ACTION OpenStopper2_action:
ST03_515_Y72_5.MoveWork:=TRUE;		(* Übergabeposition Stopper 2 *)
END_ACTION

ACTION WaitForPartOnPos3_entry:
ProcessMessage02:='';
Delay(IN:=FALSE);
END_ACTION

ACTION WaitForPartOnPos3_action:
ProcessMessage02:='2IM4';						(*warte auf Teil Übergabeposition 3*)
END_ACTION

ACTION WaitForPartOnPos3_exit:
ProcessMessage02:='';
END_ACTION

ACTION CloseStopper2_action:
ST03_515_Y72_5.MoveInit:=TRUE;		(* Übergabeposition Stopper 2 *)
END_ACTION

ACTION OpenStopper3_action:
ST03_515_Y72_6.MoveWork:=TRUE;		(* Übergabeposition Stopper 3 *)
END_ACTION

ACTION WaitForPartOnPos4_entry:
ProcessMessage02:='';
Delay(IN:=FALSE);
END_ACTION

ACTION WaitForPartOnPos4_action:
ProcessMessage02:='2IM3';						(*warte auf Teil Übergabeposition 4*)
Delay(
	IN:=NOT ST03_513_B70_7.BitInToCheck AND	(* ISK auf Übergabeposition  1*)
		NOT ST03_514_B71_2.BitInToCheck AND	(* ISK auf Übergabeposition  2*)
		NOT ST03_514_B71_5.BitInToCheck AND	(* ISK auf Übergabeposition  3*)
		NOT ST03_514_B71_6.BitInToCheck		(* ISK auf Übergabeposition  4*),
	PT:=t#1s);
END_ACTION

ACTION WaitForPartOnPos4_exit:
ProcessMessage02:='';
Delay(IN:=FALSE);
END_ACTION

ACTION CloseStopper3_action:
ST03_515_Y72_6.MoveInit:=TRUE;		(* Übergabeposition Stopper 3 *)
END_ACTION

ACTION SeqEnd_action:
SFCTime:=TIME_TO_DINT(TIME()-SFCTimeStart);
State:=STATE_WAIT;
END_ACTION

TRANSITION .ActualArea:
Robot01.ActualArea <> 4
END_TRANSITION

TRANSITION Check_Part:
NOT ST03_513_B70_7.BitInToCheck OR	(* ISK auf Übergabeposition  1*)
NOT ST03_514_B71_2.BitInToCheck OR	(* ISK auf Übergabeposition  2*)
NOT ST03_514_B71_5.BitInToCheck OR	(* ISK auf Übergabeposition  3*)
NOT ST03_514_B71_6.BitInToCheck		(* ISK auf Übergabeposition  4*)
END_TRANSITION

TRANSITION PosEmpty:
NOT ST03_513_B70_4.BitInToCheck			 	(*  ISK anwesend am Stopper*)
END_TRANSITION

TRANSITION State Ok:
ST03_515_Y72_2.State=STATE_OK (* Führungsschiene  Zuführung Vereinzler AST/GST *)
END_TRANSITION

TRANSITION Part Ready:
ST03_513_B70_4.BitInToCheck	(*  ISK anwesend am Stopper*)
END_TRANSITION

TRANSITION PosFull:
ST03_513_B70_4.BitInToCheck			 	(*  ISK anwesend am Stopper*)
END_TRANSITION

TRANSITION State Ok:
ST03_515_Y72_2.State=STATE_OK (* Führungsschiene  Zuführung Vereinzler AST/GST *)
END_TRANSITION

TRANSITION Pos1Empty:
NOT ST03_513_B70_7.BitInToCheck AND 	(*  ISK auf Übergabeposition 1*)
Robot01.ActualArea <> 4
END_TRANSITION

TRANSITION State Ok:
ST03_515_Y72_3.State=STATE_OK 	(* Führungsschiene  Zuführung Stopper AST/GST *)
END_TRANSITION

TRANSITION Pos1 Ready:
ST03_513_B70_7.BitInToCheck 		 (* ISK auf Übergabeposition 1 *)
END_TRANSITION

TRANSITION Pos1Full:
ST03_513_B70_7.BitInToCheck 	(*  ISK auf Übergabeposition 1*)
END_TRANSITION

TRANSITION State Ok:
ST03_515_Y72_3.State=STATE_OK AND 	(* Führungsschiene  Zuführung Stopper AST/GST *)
ST03_515_Y72_2.State=STATE_OK (* Führungsschiene  Zuführung Vereinzler AST/GST *)
END_TRANSITION

TRANSITION Pos2Empty:
NOT ST03_514_B71_2.BitInToCheck  	(*  ISK auf Übergabeposition 2*)
END_TRANSITION

TRANSITION State Ok:
ST03_515_Y72_4.State=STATE_OK 	(* Übergabeposition Stopper 1 AST/GST *)
END_TRANSITION

TRANSITION Pos3Full:
ST03_514_B71_5.BitInToCheck	 	(*  ISK auf Übergabeposition 3*)
END_TRANSITION

TRANSITION Pos3Empty:
NOT ST03_514_B71_5.BitInToCheck  	(*  ISK auf Übergabeposition 3*)
END_TRANSITION

TRANSITION Pos2 Ready:
ST03_514_B71_2.BitInToCheck 		 (* ISK auf Übergabeposition 2 *)
END_TRANSITION

TRANSITION Pos2Full:
ST03_514_B71_2.BitInToCheck	 	(*  ISK auf Übergabeposition 2*)
END_TRANSITION

TRANSITION State Ok:
ST03_515_Y72_4.State=STATE_OK 	(* Übergabeposition Stopper 1 AST/GST *)
END_TRANSITION

TRANSITION Pos3Empty:
NOT ST03_514_B71_5.BitInToCheck  	(*  ISK auf Übergabeposition 3*)
END_TRANSITION

TRANSITION State Ok:
ST03_515_Y72_5.State=STATE_OK 	(* Übergabeposition Stopper 2 AST/GST *)
END_TRANSITION

TRANSITION Po4Full:
ST03_514_B71_6.BitInToCheck 		(*  ISK auf Übergabeposition 4*)
END_TRANSITION

TRANSITION Pos4Empty:
NOT ST03_514_B71_6.BitInToCheck  	(*  ISK auf Übergabeposition 4*)
END_TRANSITION

TRANSITION Pos3 Ready:
ST03_514_B71_5.BitInToCheck 	 (* ISK auf Übergabeposition 3 *)
END_TRANSITION

TRANSITION Pos3Full:
ST03_514_B71_5.BitInToCheck	 	(*  ISK auf Übergabeposition 3*)
END_TRANSITION

TRANSITION State Ok:
ST03_515_Y72_5.State=STATE_OK 	(* Übergabeposition Stopper 2 AST/GST *)
END_TRANSITION

TRANSITION Pos4Empty:
NOT ST03_514_B71_6.BitInToCheck  	(*  ISK auf Übergabeposition 4*)
END_TRANSITION

TRANSITION State Ok:
ST03_515_Y72_6.State=STATE_OK 	(* Übergabeposition Stopper 3 AST/GST *)
END_TRANSITION

TRANSITION Pos4 Ready:
ST03_514_B71_6.BitInToCheck  OR		 (* ISK auf Übergabeposition 4 *)
Delay.Q
END_TRANSITION

TRANSITION Po4Full:
ST03_514_B71_6.BitInToCheck 		(*  ISK auf Übergabeposition 4*)
END_TRANSITION

TRANSITION State Ok:
ST03_515_Y72_6.State=STATE_OK 	(* Übergabeposition Stopper 3 AST/GST *)
END_TRANSITION
END_PROGRAM

(* POU Stations/ST_03_Ruestsaetze/ST_03_SFCs/Zufuehrungen/ST03_7pol_Wendeeinheit, SFC *)
 PROGRAM ST03_7pol_Wendeeinheit
VAR_OUTPUT
	SFCCurrentPOU			: STRING:='ST03_7pol_Wendeeinheit';
	SFCCurrentStep			: STRING:='';
	FB_CurrentStepHistorie	: FB_CurrentStepHistorie;
	SFCTime					: DINT;
	State   				: StateObject	:= STATE_WAIT;
	Result  				: StateResult;
END_VAR
VAR_INPUT
	Start				:BOOL;
END_VAR
VAR
	MsgOK				: BOOL;
	MsgCancel			: BOOL;
	SFCRun				: BOOL;
	SFCTimeStart		: TIME;
	Delay				: TON;
	(* Userdefinded area *)
	WenderDone			: BOOL;
	OverrideHelp			:DINT;
END_VAR
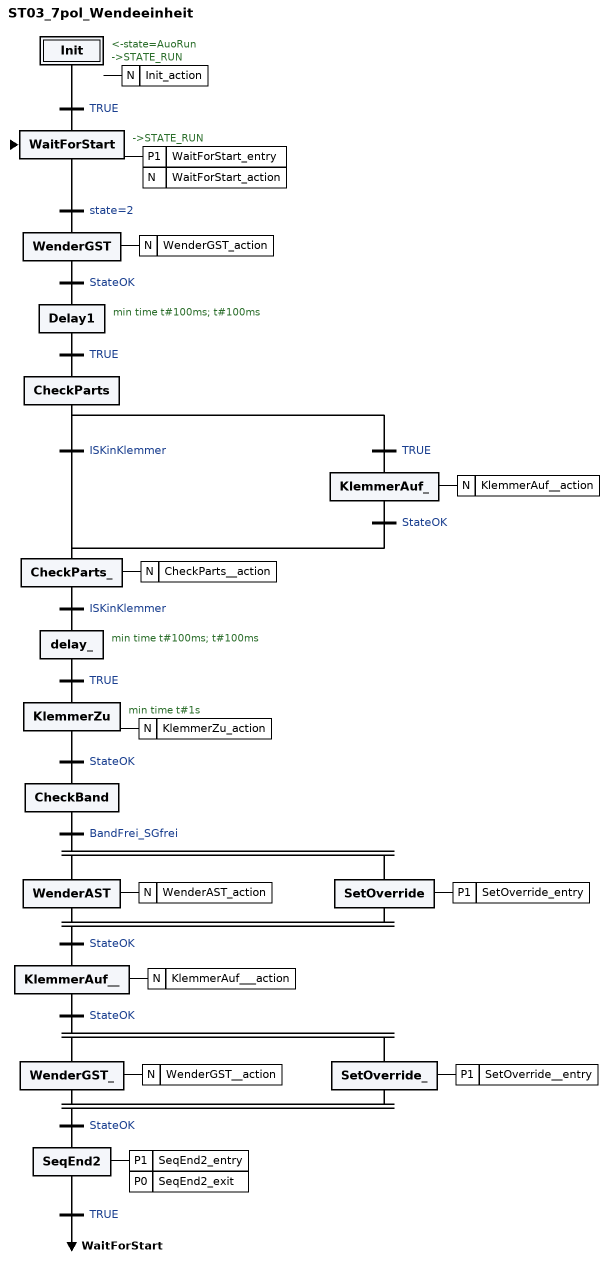
INITIAL_STEP Init: (* <-state=AuoRun / ->STATE_RUN *)
	Init_action(N);
END_STEP
TRANSITION FROM Init TO WaitForStart := TRUE;
END_TRANSITION
STEP WaitForStart: (* ->STATE_RUN *)
	WaitForStart_entry(P1);
	WaitForStart_action(N);
END_STEP
TRANSITION FROM WaitForStart TO WenderGST := state=2;
END_TRANSITION
STEP WenderGST:
	WenderGST_action(N);
END_STEP
TRANSITION FROM WenderGST TO Delay1 := StateOK;
END_TRANSITION
STEP Delay1: (* min time t#100ms; t#100ms *)
END_STEP
TRANSITION FROM Delay1 TO CheckParts := TRUE;
END_TRANSITION
STEP CheckParts:
END_STEP
TRANSITION FROM CheckParts TO CheckParts_ := ISKinKlemmer;
END_TRANSITION
TRANSITION FROM CheckParts TO KlemmerAuf_ := TRUE;
END_TRANSITION
STEP KlemmerAuf_:
	KlemmerAuf__action(N);
END_STEP
TRANSITION FROM KlemmerAuf_ TO CheckParts_ := StateOK;
END_TRANSITION
STEP CheckParts_:
	CheckParts__action(N);
END_STEP
TRANSITION FROM CheckParts_ TO delay_ := ISKinKlemmer;
END_TRANSITION
STEP delay_: (* min time t#100ms; t#100ms *)
END_STEP
TRANSITION FROM delay_ TO KlemmerZu := TRUE;
END_TRANSITION
STEP KlemmerZu: (* min time t#1s *)
	KlemmerZu_action(N);
END_STEP
TRANSITION FROM KlemmerZu TO CheckBand := StateOK;
END_TRANSITION
STEP CheckBand:
END_STEP
TRANSITION FROM CheckBand TO (WenderAST, SetOverride) := BandFrei_SGfrei;
END_TRANSITION
STEP WenderAST:
	WenderAST_action(N);
END_STEP
STEP SetOverride:
	SetOverride_entry(P1);
END_STEP
TRANSITION FROM (WenderAST, SetOverride) TO KlemmerAuf__ := StateOK;
END_TRANSITION
STEP KlemmerAuf__:
	KlemmerAuf___action(N);
END_STEP
TRANSITION FROM KlemmerAuf__ TO (WenderGST_, SetOverride_) := StateOK;
END_TRANSITION
STEP WenderGST_:
	WenderGST__action(N);
END_STEP
STEP SetOverride_:
	SetOverride__entry(P1);
END_STEP
TRANSITION FROM (WenderGST_, SetOverride_) TO SeqEnd2 := StateOK;
END_TRANSITION
STEP SeqEnd2:
	SeqEnd2_entry(P1);
	SeqEnd2_exit(P0);
END_STEP
TRANSITION FROM SeqEnd2 TO WaitForStart := TRUE;
END_TRANSITION

ACTION Init_action:
Start:=FALSE;
State:=STATE_WAIT;
MsgOK:=FALSE;
MsgCancel:=FALSE;
SFCRun:=FALSE;
Result:=RESULT_NON;
IF 	OverrideHelp <> 0 THEN
	MP.ST02.Override_Band:=OverrideHelp;
END_IF
END_ACTION

ACTION WaitForStart_entry:
;
END_ACTION

ACTION WaitForStart_action:
IF 	Start   THEN
	State:=STATE_RUN;
	Result:=RESULT_NON;
	SFCTimeStart:=TIME();
	Start:=FALSE;
	WenderDone:=FALSE;
ELSE
	State:=STATE_WAIT;
	MsgOK:=FALSE;
	MsgCancel:=FALSE;
	SFCRun:=FALSE;
END_IF
END_ACTION

ACTION WenderGST_action:
ST03_515_Y72_1.MoveInit:=TRUE;		(* Rinne schwenkern AST/GST *)
END_ACTION

ACTION KlemmerAuf__action:
ST03_515_Y72_0.MoveInit:=TRUE;		(* ISK Klemmer AST/GST *)
END_ACTION

ACTION CheckParts__action:
ProcessMessage01:='1IM6';						(*'warte auf Teil in Vereinzelung*)
END_ACTION

ACTION KlemmerZu_action:
ST03_515_Y72_0.MoveWork:=TRUE;		(* ISK Klemmer AST/GST *)
END_ACTION

ACTION WenderAST_action:
ST03_515_Y72_1.MoveWork:=TRUE;		(* Rinne schwenkern AST/GST *)
END_ACTION

ACTION SetOverride_entry:
IF 	MP.ST02.Override_Band > 10 THEN
	OverrideHelp:=MP.ST02.Override_Band;
	MP.ST02.Override_Band:= 0;
END_IF
END_ACTION

ACTION KlemmerAuf___action:
ST03_515_Y72_0.MoveInit:=TRUE;
END_ACTION

ACTION WenderGST__action:
ST03_515_Y72_1.MoveInit:=TRUE;		(* Rinne schwenkern AST/GST *)
END_ACTION

ACTION SetOverride__entry:
MP.ST02.Override_Band:=OverrideHelp;
END_ACTION

ACTION SeqEnd2_entry:
WenderDone:=TRUE;
END_ACTION

ACTION SeqEnd2_exit:
WenderDone:=FALSE;
END_ACTION

TRANSITION StateOK:
ST03_515_Y72_1.State = STATE_OK			 (* Rinne schwenkern AST/GST *)
AND gTipImp
END_TRANSITION

TRANSITION ISKinKlemmer:
ST03_512_XG1.BitInToCheck 	(* ISK in Klemmer *)
AND gTipImp
END_TRANSITION

TRANSITION StateOK:
ST03_515_Y72_0.State = STATE_OK		(*   ISK Klemmer AST/GST *)
AND gTipImp
END_TRANSITION

TRANSITION ISKinKlemmer:
ST03_512_XG1.BitInToCheck AND 	(* ISK in Klemmer *)
gTipImp
END_TRANSITION

TRANSITION StateOK:
ST03_515_Y72_0.State = STATE_OK			(* ISK Klemmer AST/GST *)
AND gTipImp
END_TRANSITION

TRANSITION BandFrei_SGfrei:
ST03_514_B71_7.BitInToCheck  	(* Führungsschiene frei zum schwenken *)
AND (ST00_73_K4.BitInToCheck OR ST02_S1_40K01.BitInToCheck)		(*Schnittstelle Freigabe von Spritzmaschine (nur für Anlagen ohne Rundtisch)*)
AND gTipImp
END_TRANSITION

TRANSITION StateOK:
ST03_515_Y72_1.State = STATE_OK 	(* Förderband  Zuführung Vereinzelner Wender AST/GST *)
AND gTipImp
END_TRANSITION

TRANSITION StateOK:
ST03_515_Y72_0.State = STATE_OK	(* ISK Klemmer AST/GST *)
AND gTipImp
END_TRANSITION

TRANSITION StateOK:
ST03_515_Y72_1.State = STATE_OK 	(* Rinne schwenkern AST/GST *)
AND gTipImp
END_TRANSITION
END_PROGRAM

(* POU Stations/ST_03_Ruestsaetze/ST_03_SFCs/Zufuehrungen/ST03_9pol_Wendeeinheit, SFC *)
 PROGRAM ST03_9pol_Wendeeinheit
VAR_OUTPUT
	SFCCurrentPOU			: STRING:='ST03_7pol_Wendeeinheit';
	SFCCurrentStep			: STRING:='';
	FB_CurrentStepHistorie	: FB_CurrentStepHistorie;
	SFCTime					: DINT;
	State   				: StateObject	:= STATE_WAIT;
	Result  				: StateResult;
END_VAR
VAR_INPUT
	Start				:BOOL;
END_VAR
VAR
	MsgOK				: BOOL;
	MsgCancel			: BOOL;
	SFCRun				: BOOL;
	SFCTimeStart		: TIME;
	Delay				: TON;
	(* Userdefinded area *)
	WenderDone			: BOOL;
	OverrideHelp			:DINT;
END_VAR
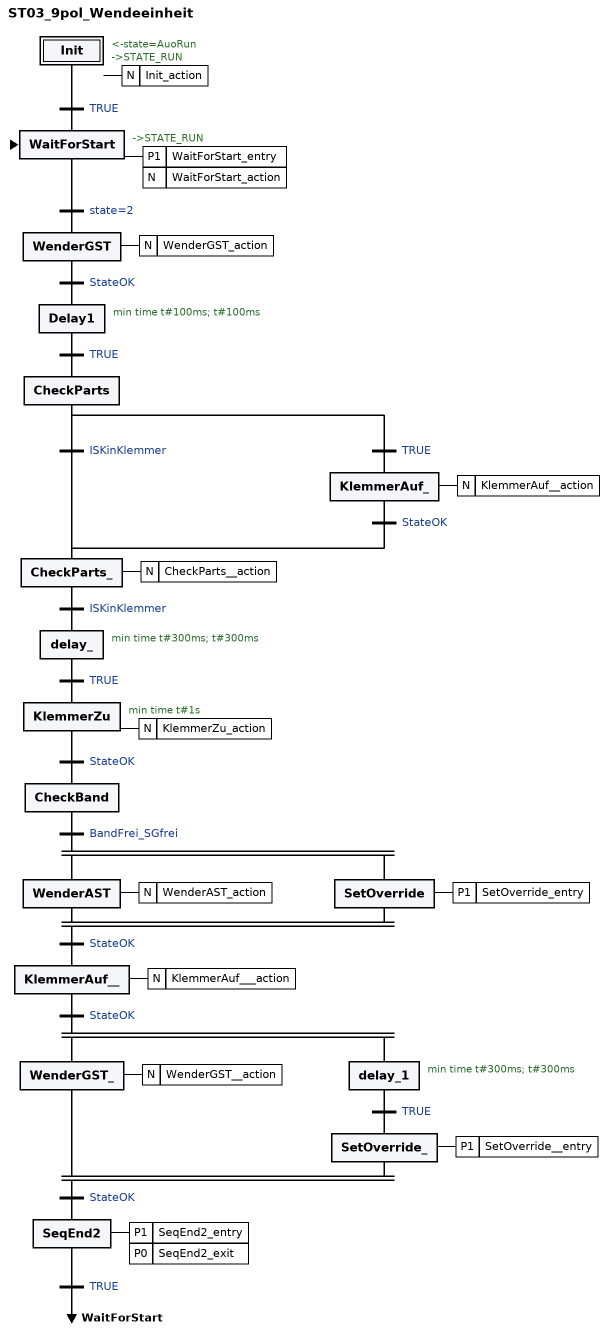
INITIAL_STEP Init: (* <-state=AuoRun / ->STATE_RUN *)
	Init_action(N);
END_STEP
TRANSITION FROM Init TO WaitForStart := TRUE;
END_TRANSITION
STEP WaitForStart: (* ->STATE_RUN *)
	WaitForStart_entry(P1);
	WaitForStart_action(N);
END_STEP
TRANSITION FROM WaitForStart TO WenderGST := state=2;
END_TRANSITION
STEP WenderGST:
	WenderGST_action(N);
END_STEP
TRANSITION FROM WenderGST TO Delay1 := StateOK;
END_TRANSITION
STEP Delay1: (* min time t#100ms; t#100ms *)
END_STEP
TRANSITION FROM Delay1 TO CheckParts := TRUE;
END_TRANSITION
STEP CheckParts:
END_STEP
TRANSITION FROM CheckParts TO CheckParts_ := ISKinKlemmer;
END_TRANSITION
TRANSITION FROM CheckParts TO KlemmerAuf_ := TRUE;
END_TRANSITION
STEP KlemmerAuf_:
	KlemmerAuf__action(N);
END_STEP
TRANSITION FROM KlemmerAuf_ TO CheckParts_ := StateOK;
END_TRANSITION
STEP CheckParts_:
	CheckParts__action(N);
END_STEP
TRANSITION FROM CheckParts_ TO delay_ := ISKinKlemmer;
END_TRANSITION
STEP delay_: (* min time t#300ms; t#300ms *)
END_STEP
TRANSITION FROM delay_ TO KlemmerZu := TRUE;
END_TRANSITION
STEP KlemmerZu: (* min time t#1s *)
	KlemmerZu_action(N);
END_STEP
TRANSITION FROM KlemmerZu TO CheckBand := StateOK;
END_TRANSITION
STEP CheckBand:
END_STEP
TRANSITION FROM CheckBand TO (WenderAST, SetOverride) := BandFrei_SGfrei;
END_TRANSITION
STEP WenderAST:
	WenderAST_action(N);
END_STEP
STEP SetOverride:
	SetOverride_entry(P1);
END_STEP
TRANSITION FROM (WenderAST, SetOverride) TO KlemmerAuf__ := StateOK;
END_TRANSITION
STEP KlemmerAuf__:
	KlemmerAuf___action(N);
END_STEP
TRANSITION FROM KlemmerAuf__ TO (WenderGST_, delay_1) := StateOK;
END_TRANSITION
STEP WenderGST_:
	WenderGST__action(N);
END_STEP
STEP delay_1: (* min time t#300ms; t#300ms *)
END_STEP
TRANSITION FROM delay_1 TO SetOverride_ := TRUE;
END_TRANSITION
STEP SetOverride_:
	SetOverride__entry(P1);
END_STEP
TRANSITION FROM (WenderGST_, SetOverride_) TO SeqEnd2 := StateOK;
END_TRANSITION
STEP SeqEnd2:
	SeqEnd2_entry(P1);
	SeqEnd2_exit(P0);
END_STEP
TRANSITION FROM SeqEnd2 TO WaitForStart := TRUE;
END_TRANSITION

ACTION Init_action:
Start:=FALSE;
State:=STATE_WAIT;
MsgOK:=FALSE;
MsgCancel:=FALSE;
SFCRun:=FALSE;
Result:=RESULT_NON;
IF 	OverrideHelp <> 0 THEN
	MP.ST02.Override_Band:=OverrideHelp;
END_IF
END_ACTION

ACTION WaitForStart_entry:
;
END_ACTION

ACTION WaitForStart_action:
IF 	Start   THEN
	State:=STATE_RUN;
	Result:=RESULT_NON;
	SFCTimeStart:=TIME();
	Start:=FALSE;
	WenderDone:=FALSE;
ELSE
	State:=STATE_WAIT;
	MsgOK:=FALSE;
	MsgCancel:=FALSE;
	SFCRun:=FALSE;
END_IF
END_ACTION

ACTION WenderGST_action:
ST03_515_Y72_1.MoveInit:=TRUE;		(* Rinne schwenkern AST/GST *)
END_ACTION

ACTION KlemmerAuf__action:
ST03_515_Y72_0.MoveInit:=TRUE;		(* ISK Klemmer AST/GST *)
END_ACTION

ACTION CheckParts__action:
ProcessMessage01:='1IM6';						(*'warte auf Teil in Vereinzelung*)
END_ACTION

ACTION KlemmerZu_action:
ST03_515_Y72_0.MoveWork:=TRUE;		(* ISK Klemmer AST/GST *)
END_ACTION

ACTION WenderAST_action:
ST03_515_Y72_1.MoveWork:=TRUE;		(* Rinne schwenkern AST/GST *)
END_ACTION

ACTION SetOverride_entry:
IF 	MP.ST02.Override_Band > 10 THEN
	OverrideHelp:=MP.ST02.Override_Band;
	MP.ST02.Override_Band:= 0;
END_IF
END_ACTION

ACTION KlemmerAuf___action:
ST03_515_Y72_0.MoveInit:=TRUE;
END_ACTION

ACTION WenderGST__action:
ST03_515_Y72_1.MoveInit:=TRUE;		(* Rinne schwenkern AST/GST *)
END_ACTION

ACTION SetOverride__entry:
MP.ST02.Override_Band:=OverrideHelp;
END_ACTION

ACTION SeqEnd2_entry:
WenderDone:=TRUE;
END_ACTION

ACTION SeqEnd2_exit:
WenderDone:=FALSE;
END_ACTION

TRANSITION StateOK:
ST03_515_Y72_1.State = STATE_OK			 (* Rinne schwenkern AST/GST *)
AND gTipImp
END_TRANSITION

TRANSITION ISKinKlemmer:
ST03_512_XG1.BitInToCheck 	(* ISK in Klemmer *)
AND gTipImp
END_TRANSITION

TRANSITION StateOK:
ST03_515_Y72_0.State = STATE_OK		(*   ISK Klemmer AST/GST *)
AND gTipImp
END_TRANSITION

TRANSITION ISKinKlemmer:
ST03_512_XG1.BitInToCheck AND 	(* ISK in Klemmer *)
gTipImp
END_TRANSITION

TRANSITION StateOK:
ST03_515_Y72_0.State = STATE_OK			(* ISK Klemmer AST/GST *)
AND gTipImp
END_TRANSITION

TRANSITION BandFrei_SGfrei:
ST03_514_B71_7.BitInToCheck  	(* Führungsschiene frei zum schwenken *)
AND (ST00_73_K4.BitInToCheck OR ST02_S1_40K01.BitInToCheck)		(*Schnittstelle Freigabe von Spritzmaschine (nur für Anlagen ohne Rundtisch)*)
AND gTipImp
END_TRANSITION

TRANSITION StateOK:
ST03_515_Y72_1.State = STATE_OK 	(* Förderband  Zuführung Vereinzelner Wender AST/GST *)
AND gTipImp
END_TRANSITION

TRANSITION StateOK:
ST03_515_Y72_0.State = STATE_OK	(* ISK Klemmer AST/GST *)
AND gTipImp
END_TRANSITION

TRANSITION StateOK:
ST03_515_Y72_1.State = STATE_OK 	(* Rinne schwenkern AST/GST *)
AND gTipImp
END_TRANSITION
END_PROGRAM

(* POU Stations/ST_03_Ruestsaetze/ST_03_SFCs/Zufuehrungen/ST03_88polAMG_Zufuehrung, SFC *)
 PROGRAM ST03_88polAMG_Zufuehrung
VAR_OUTPUT
	SFCCurrentPOU		: STRING:='ST03_88polAMG_Zufuehrung';
	SFCCurrentStep		: STRING:='';
	FB_CurrentStepHistorie: FB_CurrentStepHistorie;
	SFCTime				: DINT;
	State   			: StateObject	:= STATE_WAIT;
	Result  			: StateResult;
END_VAR
VAR_INPUT
	Start				:BOOL;
END_VAR
VAR
	MsgOK				: BOOL;
	MsgCancel			: BOOL;
	SFCRun				: BOOL;
	SFCTimeStart		: TIME;
	Delay				: TON;
	(* Userdefinded area *)

END_VAR
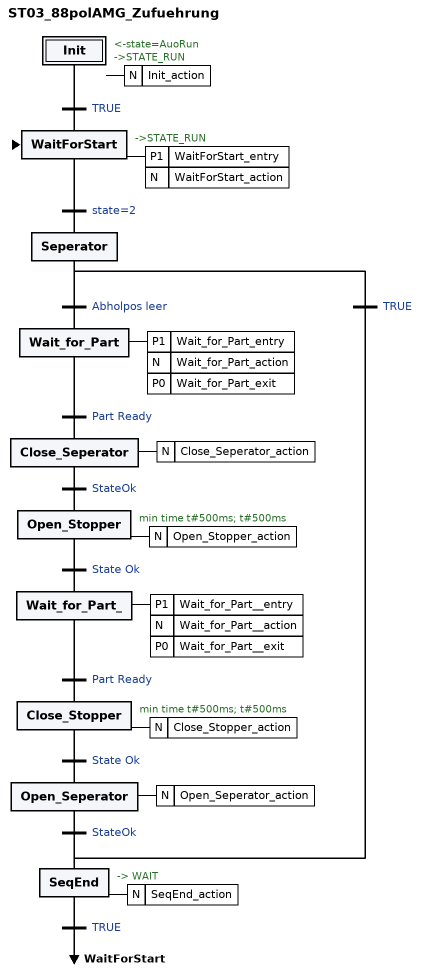
INITIAL_STEP Init: (* <-state=AuoRun / ->STATE_RUN *)
	Init_action(N);
END_STEP
TRANSITION FROM Init TO WaitForStart := TRUE;
END_TRANSITION
STEP WaitForStart: (* ->STATE_RUN *)
	WaitForStart_entry(P1);
	WaitForStart_action(N);
END_STEP
TRANSITION FROM WaitForStart TO Seperator := state=2;
END_TRANSITION
STEP Seperator:
END_STEP
TRANSITION FROM Seperator TO Wait_for_Part := Abholpos leer;
END_TRANSITION
TRANSITION FROM Seperator TO SeqEnd := TRUE;
END_TRANSITION
STEP Wait_for_Part:
	Wait_for_Part_entry(P1);
	Wait_for_Part_action(N);
	Wait_for_Part_exit(P0);
END_STEP
TRANSITION FROM Wait_for_Part TO Close_Seperator := Part Ready;
END_TRANSITION
STEP Close_Seperator:
	Close_Seperator_action(N);
END_STEP
TRANSITION FROM Close_Seperator TO Open_Stopper := StateOk;
END_TRANSITION
STEP Open_Stopper: (* min time t#500ms; t#500ms *)
	Open_Stopper_action(N);
END_STEP
TRANSITION FROM Open_Stopper TO Wait_for_Part_ := State Ok;
END_TRANSITION
STEP Wait_for_Part_:
	Wait_for_Part__entry(P1);
	Wait_for_Part__action(N);
	Wait_for_Part__exit(P0);
END_STEP
TRANSITION FROM Wait_for_Part_ TO Close_Stopper := Part Ready;
END_TRANSITION
STEP Close_Stopper: (* min time t#500ms; t#500ms *)
	Close_Stopper_action(N);
END_STEP
TRANSITION FROM Close_Stopper TO Open_Seperator := State Ok;
END_TRANSITION
STEP Open_Seperator:
	Open_Seperator_action(N);
END_STEP
TRANSITION FROM Open_Seperator TO SeqEnd := StateOk;
END_TRANSITION
STEP SeqEnd: (* -> WAIT *)
	SeqEnd_action(N);
END_STEP
TRANSITION FROM SeqEnd TO WaitForStart := TRUE;
END_TRANSITION

ACTION Init_action:
Start:=FALSE;
State:=STATE_WAIT;
MsgOK:=FALSE;
MsgCancel:=FALSE;
SFCRun:=FALSE;
Result:=RESULT_NON;
END_ACTION

ACTION WaitForStart_entry:
;
END_ACTION

ACTION WaitForStart_action:
IF 	Start   THEN
	State:=STATE_RUN;
	Result:=RESULT_NON;
	SFCTimeStart:=TIME();
	Start:=FALSE;
ELSE
	State:=STATE_WAIT;
	MsgOK:=FALSE;
	MsgCancel:=FALSE;
	SFCRun:=FALSE;
END_IF
END_ACTION

ACTION Wait_for_Part_entry:
ProcessMessage01:='';
Delay.IN:=FALSE;
Delay();
END_ACTION

ACTION Wait_for_Part_action:
ProcessMessage01:='1IM9';(*warte auf Teil in Stopper*)
Delay.IN:=ST03_521_B69_6.BitInToCheck; 		(*  ISK an stopper.*)
Delay.PT:=T#500ms;
Delay();
END_ACTION

ACTION Wait_for_Part_exit:
ProcessMessage01:='';
END_ACTION

ACTION Close_Seperator_action:
ST03_522_Y70_1.MoveWork:=TRUE;		(* Zuführung Vereinzler AST/GST *)
END_ACTION

ACTION Open_Stopper_action:
ST03_522_Y70_2.MoveWork:=TRUE;		(* Züführung Stopper AST/GST *)
END_ACTION

ACTION Wait_for_Part__entry:
ProcessMessage01:='';
Delay.IN:=FALSE;
Delay();
END_ACTION

ACTION Wait_for_Part__action:
ProcessMessage01:='1IM10';(*warte auf Teil in Abholposition*)
Delay.IN:=	ST03_Init_AbholPos.RoboPos31 OR
			ST03_Init_AbholPos.RoboPos35;
Delay.PT:=T#500ms;
Delay();
END_ACTION

ACTION Wait_for_Part__exit:
ProcessMessage01:='';
END_ACTION

ACTION Close_Stopper_action:
ST03_522_Y70_2.MoveInit:=TRUE;		(* Züführung Stopper AST/GST *)
END_ACTION

ACTION Open_Seperator_action:
ST03_522_Y70_1.MoveInit:=TRUE;		(* Zuführung Vereinzler AST/GST *)
END_ACTION

ACTION SeqEnd_action:
SFCTime:=TIME_TO_DINT(TIME()-SFCTimeStart);
State:=STATE_WAIT;
END_ACTION

TRANSITION Abholpos leer:
NOT  ST03_521_B69_7.BitInToCheck AND		(*  ISK Lageerkennung links*)
NOT  ST03_522_B70_0.BitInToCheck 		(*  ISK Lageerkennung rechts*)
END_TRANSITION

TRANSITION Part Ready:
Delay.Q AND
NOT ST03_521_B69_7.BitInToCheck	AND		(*  ISK Lageerkennung links*)
NOT ST03_522_B70_0.BitInToCheck	AND		(*  ISK Lageerkennung rechts*)
ST03_521_B69_6.BitInToCheck	AND				(*  ISK anwesend am Stoper*)
Robot01.ActualArea <> 4
END_TRANSITION

TRANSITION StateOk:
ST03_522_Y70_1.State=STATE_OK 	(* Zuführung Vereinzler AST/GST *)
END_TRANSITION

TRANSITION State Ok:
ST03_522_Y70_2.State=STATE_OK 	(* Züführung Stopper AST/GST *)
END_TRANSITION

TRANSITION Part Ready:
Delay.Q AND
Robot01.ActualArea <> 4
END_TRANSITION

TRANSITION State Ok:
ST03_522_Y70_2.State=STATE_OK 	(*Züführung Stopper AST/GST *)
END_TRANSITION

TRANSITION StateOk:
ST03_522_Y70_1.State=STATE_OK 	(* Zuführung Vereinzler AST/GST *)
END_TRANSITION
END_PROGRAM

(* POU Stations/ST_03_Ruestsaetze/ST_03_SFCs/Zufuehrungen/ST03_120pol_Zufuehrung, SFC *)
 PROGRAM ST03_120pol_Zufuehrung
VAR_OUTPUT
	SFCCurrentPOU		: STRING:='ST03_120pol_Zufuehrung';
	SFCCurrentStep		: STRING:='';
	FB_CurrentStepHistorie: FB_CurrentStepHistorie;
	SFCTime				: DINT;
	State   			: StateObject	:= STATE_WAIT;
	Result  			: StateResult;
END_VAR
VAR_INPUT
	Start				:BOOL;
END_VAR
VAR
	MsgOK				: BOOL;
	MsgCancel			: BOOL;
	SFCRun				: BOOL;
	SFCTimeStart		: TIME;
	Delay				: TON;
	(* Userdefinded area *)

END_VAR
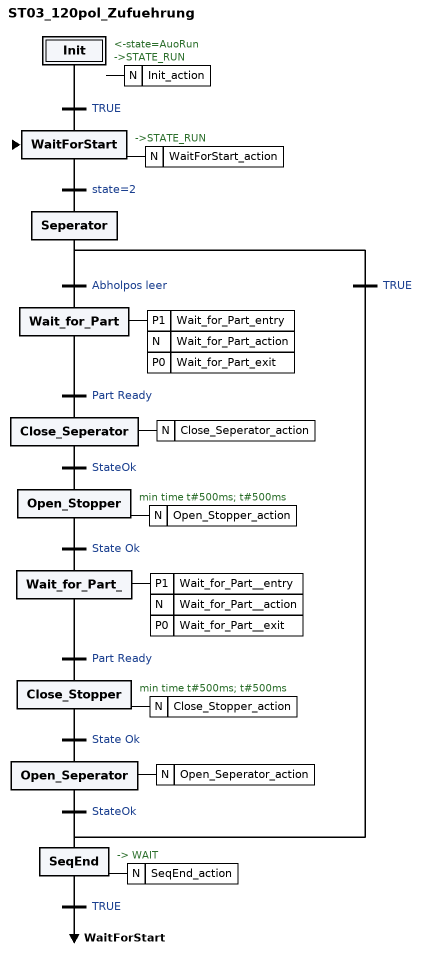
INITIAL_STEP Init: (* <-state=AuoRun / ->STATE_RUN *)
	Init_action(N);
END_STEP
TRANSITION FROM Init TO WaitForStart := TRUE;
END_TRANSITION
STEP WaitForStart: (* ->STATE_RUN *)
	WaitForStart_action(N);
END_STEP
TRANSITION FROM WaitForStart TO Seperator := state=2;
END_TRANSITION
STEP Seperator:
END_STEP
TRANSITION FROM Seperator TO Wait_for_Part := Abholpos leer;
END_TRANSITION
TRANSITION FROM Seperator TO SeqEnd := TRUE;
END_TRANSITION
STEP Wait_for_Part:
	Wait_for_Part_entry(P1);
	Wait_for_Part_action(N);
	Wait_for_Part_exit(P0);
END_STEP
TRANSITION FROM Wait_for_Part TO Close_Seperator := Part Ready;
END_TRANSITION
STEP Close_Seperator:
	Close_Seperator_action(N);
END_STEP
TRANSITION FROM Close_Seperator TO Open_Stopper := StateOk;
END_TRANSITION
STEP Open_Stopper: (* min time t#500ms; t#500ms *)
	Open_Stopper_action(N);
END_STEP
TRANSITION FROM Open_Stopper TO Wait_for_Part_ := State Ok;
END_TRANSITION
STEP Wait_for_Part_:
	Wait_for_Part__entry(P1);
	Wait_for_Part__action(N);
	Wait_for_Part__exit(P0);
END_STEP
TRANSITION FROM Wait_for_Part_ TO Close_Stopper := Part Ready;
END_TRANSITION
STEP Close_Stopper: (* min time t#500ms; t#500ms *)
	Close_Stopper_action(N);
END_STEP
TRANSITION FROM Close_Stopper TO Open_Seperator := State Ok;
END_TRANSITION
STEP Open_Seperator:
	Open_Seperator_action(N);
END_STEP
TRANSITION FROM Open_Seperator TO SeqEnd := StateOk;
END_TRANSITION
STEP SeqEnd: (* -> WAIT *)
	SeqEnd_action(N);
END_STEP
TRANSITION FROM SeqEnd TO WaitForStart := TRUE;
END_TRANSITION

ACTION Init_action:
Start:=FALSE;
State:=STATE_WAIT;
MsgOK:=FALSE;
MsgCancel:=FALSE;
SFCRun:=FALSE;
Result:=RESULT_NON;
END_ACTION

ACTION WaitForStart_action:
IF 	Start   THEN
	State:=STATE_RUN;
	Result:=RESULT_NON;
	SFCTimeStart:=TIME();
	Start:=FALSE;
ELSE
	State:=STATE_WAIT;
	MsgOK:=FALSE;
	MsgCancel:=FALSE;
	SFCRun:=FALSE;
END_IF
END_ACTION

ACTION Wait_for_Part_entry:
ProcessMessage01:='';
Delay.IN:=FALSE;
Delay();
END_ACTION

ACTION Wait_for_Part_action:
ProcessMessage01:='1IM9';(*warte auf Teil in Stopper*)
Delay.IN:=ST03_531_B69_6.BitInToCheck; 		(*  ISK an stopper.*)
Delay.PT:=T#500ms;
Delay();
END_ACTION

ACTION Wait_for_Part_exit:
ProcessMessage01:='';
END_ACTION

ACTION Close_Seperator_action:
ST03_532_Y70_1.MoveWork:=TRUE;		(*Zuführung Vereinzler AST/GST *)
END_ACTION

ACTION Open_Stopper_action:
ST03_532_Y70_2.MoveWork:=TRUE;		(* Züführung Stopper AST/GST *)
END_ACTION

ACTION Wait_for_Part__entry:
ProcessMessage01:='';
Delay.IN:=FALSE;
Delay();
END_ACTION

ACTION Wait_for_Part__action:
ProcessMessage01:='1IM10';(*warte auf Teil in Abholposition*)
Delay.IN:=	ST03_Init_AbholPos.RoboPos31 OR
			ST03_Init_AbholPos.RoboPos35;
Delay.PT:=T#500ms;
Delay();
END_ACTION

ACTION Wait_for_Part__exit:
ProcessMessage01:='';
END_ACTION

ACTION Close_Stopper_action:
ST03_532_Y70_2.MoveInit:=TRUE;		(* Züführung Stopper AST/GST *)
END_ACTION

ACTION Open_Seperator_action:
ST03_532_Y70_1.MoveInit:=TRUE;		(* Zuführung Vereinzler AST/GST *)
END_ACTION

ACTION SeqEnd_action:
SFCTime:=TIME_TO_DINT(TIME()-SFCTimeStart);
State:=STATE_WAIT;
END_ACTION

TRANSITION Abholpos leer:
NOT  ST03_531_B69_7.BitInToCheck AND	(*ISK rechts Lageerkennung*)
NOT ST03_532_B70_0.BitInToCheck		(*ISK links Lageerkennung*)
END_TRANSITION

TRANSITION Part Ready:
Delay.Q AND
NOT ST03_531_B69_7.BitInToCheck	AND		(*ISK rechts Lageerkennung*)
NOT ST03_532_B70_0.BitInToCheck	AND		(*ISK links Lageerkennung*)
ST03_531_B69_6.BitInToCheck	AND			(*ISK anwesend am Stoper*)
Robot01.ActualArea <> 4
END_TRANSITION

TRANSITION StateOk:
ST03_532_Y70_1.State=STATE_OK 	(* Zuführung Vereinzler AST/GST *)
END_TRANSITION

TRANSITION State Ok:
ST03_532_Y70_2.State=STATE_OK 	(* Züführung Stopper AST/GST *)
END_TRANSITION

TRANSITION Part Ready:
Delay.Q AND
Robot01.ActualArea <> 4
END_TRANSITION

TRANSITION State Ok:
ST03_532_Y70_2.State=STATE_OK 	(*Züführung Stopper AST/GST *)
END_TRANSITION

TRANSITION StateOk:
ST03_532_Y70_1.State=STATE_OK 	(* Zuführung Vereinzler AST/GST *)
END_TRANSITION
END_PROGRAM

(* POU Stations/ST_03_Ruestsaetze/ST_03_SFCs/Zufuehrungen/ST03_21pol_Zufuehrung, SFC *)
 PROGRAM ST03_21pol_Zufuehrung
VAR_OUTPUT
	SFCCurrentPOU		: STRING:='ST03_21pol_Zufuehrung';
	SFCCurrentStep		: STRING:='';
	FB_CurrentStepHistorie: FB_CurrentStepHistorie;
	SFCTime				: DINT;
	State   			: StateObject	:= STATE_WAIT;
	Result  			: StateResult;
END_VAR
VAR_INPUT
	Start				:BOOL;
END_VAR
VAR
	MsgOK				: BOOL;
	MsgCancel			: BOOL;
	SFCRun				: BOOL;
	SFCTimeStart		: TIME;
	Delay				: TON;
	(* Userdefinded area *)

END_VAR
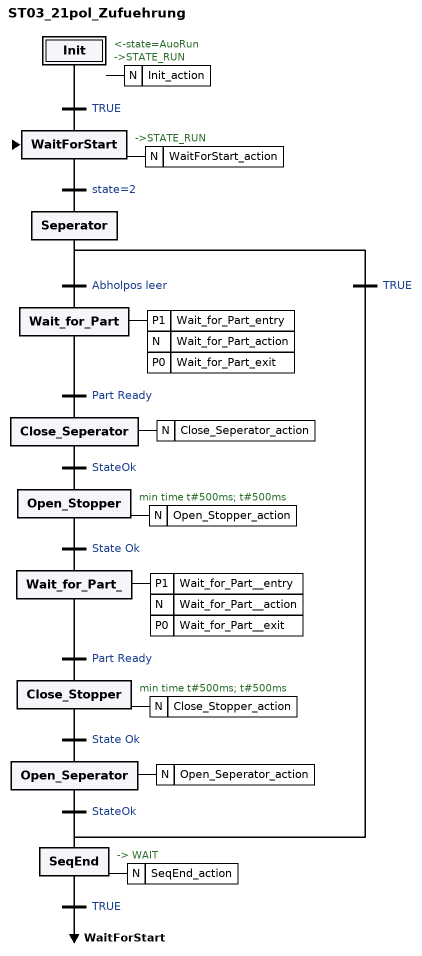
INITIAL_STEP Init: (* <-state=AuoRun / ->STATE_RUN *)
	Init_action(N);
END_STEP
TRANSITION FROM Init TO WaitForStart := TRUE;
END_TRANSITION
STEP WaitForStart: (* ->STATE_RUN *)
	WaitForStart_action(N);
END_STEP
TRANSITION FROM WaitForStart TO Seperator := state=2;
END_TRANSITION
STEP Seperator:
END_STEP
TRANSITION FROM Seperator TO Wait_for_Part := Abholpos leer;
END_TRANSITION
TRANSITION FROM Seperator TO SeqEnd := TRUE;
END_TRANSITION
STEP Wait_for_Part:
	Wait_for_Part_entry(P1);
	Wait_for_Part_action(N);
	Wait_for_Part_exit(P0);
END_STEP
TRANSITION FROM Wait_for_Part TO Close_Seperator := Part Ready;
END_TRANSITION
STEP Close_Seperator:
	Close_Seperator_action(N);
END_STEP
TRANSITION FROM Close_Seperator TO Open_Stopper := StateOk;
END_TRANSITION
STEP Open_Stopper: (* min time t#500ms; t#500ms *)
	Open_Stopper_action(N);
END_STEP
TRANSITION FROM Open_Stopper TO Wait_for_Part_ := State Ok;
END_TRANSITION
STEP Wait_for_Part_:
	Wait_for_Part__entry(P1);
	Wait_for_Part__action(N);
	Wait_for_Part__exit(P0);
END_STEP
TRANSITION FROM Wait_for_Part_ TO Close_Stopper := Part Ready;
END_TRANSITION
STEP Close_Stopper: (* min time t#500ms; t#500ms *)
	Close_Stopper_action(N);
END_STEP
TRANSITION FROM Close_Stopper TO Open_Seperator := State Ok;
END_TRANSITION
STEP Open_Seperator:
	Open_Seperator_action(N);
END_STEP
TRANSITION FROM Open_Seperator TO SeqEnd := StateOk;
END_TRANSITION
STEP SeqEnd: (* -> WAIT *)
	SeqEnd_action(N);
END_STEP
TRANSITION FROM SeqEnd TO WaitForStart := TRUE;
END_TRANSITION

ACTION Init_action:
Start:=FALSE;
State:=STATE_WAIT;
MsgOK:=FALSE;
MsgCancel:=FALSE;
SFCRun:=FALSE;
Result:=RESULT_NON;
END_ACTION

ACTION WaitForStart_action:
IF 	Start   THEN
	State:=STATE_RUN;
	Result:=RESULT_NON;
	SFCTimeStart:=TIME();
	Start:=FALSE;
ELSE
	State:=STATE_WAIT;
	MsgOK:=FALSE;
	MsgCancel:=FALSE;
	SFCRun:=FALSE;
END_IF
END_ACTION

ACTION Wait_for_Part_entry:
ProcessMessage01:='';
Delay.IN:=FALSE;
Delay();
END_ACTION

ACTION Wait_for_Part_action:
ProcessMessage01:='1IM9';(*warte auf Teil in Stopper*)
Delay.IN:=ST03_536_B69_6.BitInToCheck; 		(*  ISK an stopper.*)
Delay.PT:=T#500ms;
Delay();
END_ACTION

ACTION Wait_for_Part_exit:
ProcessMessage01:='';
END_ACTION

ACTION Close_Seperator_action:
ST03_537_Y70_1.MoveWork:=TRUE;		(*Zuführung Vereinzler AST/GST *)
END_ACTION

ACTION Open_Stopper_action:
ST03_537_Y70_2.MoveWork:=TRUE;		(* Züführung Stopper AST/GST *)
END_ACTION

ACTION Wait_for_Part__entry:
ProcessMessage01:='';
Delay.IN:=FALSE;
Delay();
END_ACTION

ACTION Wait_for_Part__action:
ProcessMessage01:='1IM10';(*warte auf Teil in Abholposition*)
Delay.IN:=	ST03_Init_AbholPos.RoboPos31 OR
			ST03_Init_AbholPos.RoboPos35;
Delay.PT:=T#500ms;
Delay();
END_ACTION

ACTION Wait_for_Part__exit:
ProcessMessage01:='';
END_ACTION

ACTION Close_Stopper_action:
ST03_537_Y70_2.MoveInit:=TRUE;		(* Züführung Stopper AST/GST *)
END_ACTION

ACTION Open_Seperator_action:
ST03_537_Y70_1.MoveInit:=TRUE;		(* Zuführung Vereinzler AST/GST *)
END_ACTION

ACTION SeqEnd_action:
SFCTime:=TIME_TO_DINT(TIME()-SFCTimeStart);
State:=STATE_WAIT;
END_ACTION

TRANSITION Abholpos leer:
NOT  ST03_536_B69_7.BitInToCheck		(*  ISK anwesend an Abholposition*)
END_TRANSITION

TRANSITION Part Ready:
Delay.Q AND
NOT ST03_536_B69_7.BitInToCheck	AND		(*ISK anwesend an Abholposition*)
NOT ST03_537_B70_0.BitInToCheck	AND		(*ISK Lageerkennung*)
ST03_536_B69_6.BitInToCheck	AND			(*ISK anwesend am Stoper*)
Robot01.ActualArea <> 4
END_TRANSITION

TRANSITION StateOk:
ST03_537_Y70_1.State=STATE_OK 	(* Zuführung Vereinzler AST/GST *)
END_TRANSITION

TRANSITION State Ok:
ST03_537_Y70_2.State=STATE_OK 	(* Züführung Stopper AST/GST *)
END_TRANSITION

TRANSITION Part Ready:
Delay.Q AND
Robot01.ActualArea <> 4
END_TRANSITION

TRANSITION State Ok:
ST03_537_Y70_2.State=STATE_OK 	(*Züführung Stopper AST/GST *)
END_TRANSITION

TRANSITION StateOk:
ST03_537_Y70_1.State=STATE_OK 	(* Zuführung Vereinzler AST/GST *)
END_TRANSITION
END_PROGRAM

(* POU Stations/ST_03_Ruestsaetze/ST_03_SFCs/Zufuehrungen/ST03_191pol_Zufuehrung, SFC *)
 PROGRAM ST03_191pol_Zufuehrung
VAR_OUTPUT
	SFCCurrentPOU		: STRING:='ST03_191pol_Zufuehrung';
	SFCCurrentStep		: STRING:='';
	FB_CurrentStepHistorie: FB_CurrentStepHistorie;
	SFCTime				: DINT;
	State   			: StateObject	:= STATE_WAIT;
	Result  			: StateResult;
END_VAR
VAR_INPUT
	Start				:BOOL;
END_VAR
VAR
	MsgOK				: BOOL;
	MsgCancel			: BOOL;
	SFCRun				: BOOL;
	SFCTimeStart		: TIME;
	Delay				: TON;
	(* Userdefinded area *)

END_VAR
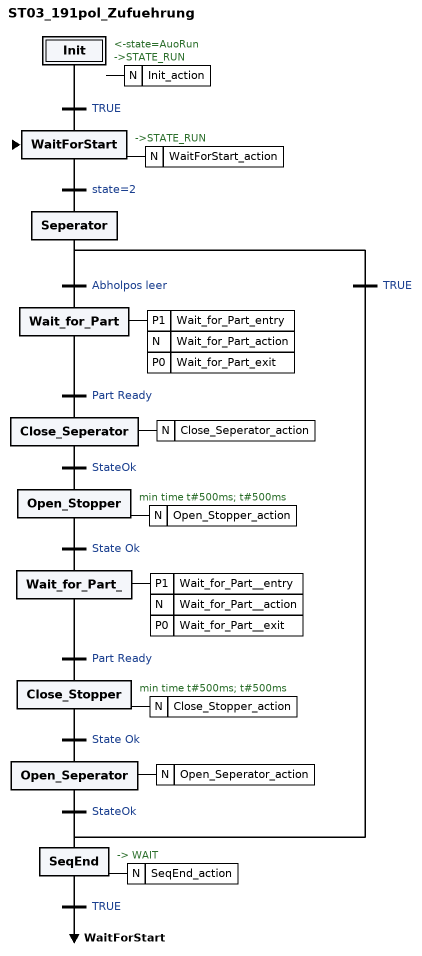
INITIAL_STEP Init: (* <-state=AuoRun / ->STATE_RUN *)
	Init_action(N);
END_STEP
TRANSITION FROM Init TO WaitForStart := TRUE;
END_TRANSITION
STEP WaitForStart: (* ->STATE_RUN *)
	WaitForStart_action(N);
END_STEP
TRANSITION FROM WaitForStart TO Seperator := state=2;
END_TRANSITION
STEP Seperator:
END_STEP
TRANSITION FROM Seperator TO Wait_for_Part := Abholpos leer;
END_TRANSITION
TRANSITION FROM Seperator TO SeqEnd := TRUE;
END_TRANSITION
STEP Wait_for_Part:
	Wait_for_Part_entry(P1);
	Wait_for_Part_action(N);
	Wait_for_Part_exit(P0);
END_STEP
TRANSITION FROM Wait_for_Part TO Close_Seperator := Part Ready;
END_TRANSITION
STEP Close_Seperator:
	Close_Seperator_action(N);
END_STEP
TRANSITION FROM Close_Seperator TO Open_Stopper := StateOk;
END_TRANSITION
STEP Open_Stopper: (* min time t#500ms; t#500ms *)
	Open_Stopper_action(N);
END_STEP
TRANSITION FROM Open_Stopper TO Wait_for_Part_ := State Ok;
END_TRANSITION
STEP Wait_for_Part_:
	Wait_for_Part__entry(P1);
	Wait_for_Part__action(N);
	Wait_for_Part__exit(P0);
END_STEP
TRANSITION FROM Wait_for_Part_ TO Close_Stopper := Part Ready;
END_TRANSITION
STEP Close_Stopper: (* min time t#500ms; t#500ms *)
	Close_Stopper_action(N);
END_STEP
TRANSITION FROM Close_Stopper TO Open_Seperator := State Ok;
END_TRANSITION
STEP Open_Seperator:
	Open_Seperator_action(N);
END_STEP
TRANSITION FROM Open_Seperator TO SeqEnd := StateOk;
END_TRANSITION
STEP SeqEnd: (* -> WAIT *)
	SeqEnd_action(N);
END_STEP
TRANSITION FROM SeqEnd TO WaitForStart := TRUE;
END_TRANSITION

ACTION Init_action:
Start:=FALSE;
State:=STATE_WAIT;
MsgOK:=FALSE;
MsgCancel:=FALSE;
SFCRun:=FALSE;
Result:=RESULT_NON;
END_ACTION

ACTION WaitForStart_action:
IF 	Start   THEN
	State:=STATE_RUN;
	Result:=RESULT_NON;
	SFCTimeStart:=TIME();
	Start:=FALSE;
ELSE
	State:=STATE_WAIT;
	MsgOK:=FALSE;
	MsgCancel:=FALSE;
	SFCRun:=FALSE;
END_IF
END_ACTION

ACTION Wait_for_Part_entry:
ProcessMessage01:='';
Delay.IN:=FALSE;
Delay();
END_ACTION

ACTION Wait_for_Part_action:
ProcessMessage01:='1IM9';(*warte auf Teil in Stopper*)
Delay.IN:=ST03_541_B69_6.BitInToCheck; 		(*  ISK an stopper.*)
Delay.PT:=T#500ms;
Delay();
END_ACTION

ACTION Wait_for_Part_exit:
ProcessMessage01:='';
END_ACTION

ACTION Close_Seperator_action:
ST03_542_Y70_1.MoveWork:=TRUE;		(*Zuführung Vereinzler AST/GST *)
END_ACTION

ACTION Open_Stopper_action:
ST03_542_Y70_2.MoveWork:=TRUE;		(* Züführung Stopper AST/GST *)
END_ACTION

ACTION Wait_for_Part__entry:
ProcessMessage01:='';
Delay.IN:=FALSE;
Delay();
END_ACTION

ACTION Wait_for_Part__action:
ProcessMessage01:='1IM10';(*warte auf Teil in Abholposition*)
Delay.IN:=	ST03_Init_AbholPos.RoboPos31 OR
			ST03_Init_AbholPos.RoboPos35;
Delay.PT:=T#500ms;
Delay();
END_ACTION

ACTION Wait_for_Part__exit:
ProcessMessage01:='';
END_ACTION

ACTION Close_Stopper_action:
ST03_542_Y70_2.MoveInit:=TRUE;		(* Züführung Stopper AST/GST *)
END_ACTION

ACTION Open_Seperator_action:
ST03_542_Y70_1.MoveInit:=TRUE;		(* Zuführung Vereinzler AST/GST *)
END_ACTION

ACTION SeqEnd_action:
SFCTime:=TIME_TO_DINT(TIME()-SFCTimeStart);
State:=STATE_WAIT;
END_ACTION

TRANSITION Abholpos leer:
NOT ST03_Init_AbholPos.RoboPos31 AND
NOT ST03_Init_AbholPos.RoboPos35
END_TRANSITION

TRANSITION Part Ready:
Delay.Q AND
NOT ST03_541_B69_7.BitInToCheck	AND		(*ISK links Lageerkennung*)
NOT ST03_542_B70_0.BitInToCheck	AND		(*ISK rechts Lageerkennung*)
ST03_541_B69_6.BitInToCheck	AND			(*ISK anwesend am Stoper*)
Robot01.ActualArea <> 4
END_TRANSITION

TRANSITION StateOk:
ST03_542_Y70_1.State=STATE_OK 	(* Zuführung Vereinzler AST/GST *)
END_TRANSITION

TRANSITION State Ok:
ST03_542_Y70_2.State=STATE_OK 	(* Züführung Stopper AST/GST *)
END_TRANSITION

TRANSITION Part Ready:
Delay.Q AND
Robot01.ActualArea <> 4
END_TRANSITION

TRANSITION State Ok:
ST03_542_Y70_2.State=STATE_OK 	(*Züführung Stopper AST/GST *)
END_TRANSITION

TRANSITION StateOk:
ST03_542_Y70_1.State=STATE_OK 	(* Zuführung Vereinzler AST/GST *)
END_TRANSITION
END_PROGRAM

(* POU Stations/ST_03_Ruestsaetze/ST_03_SFCs/Zufuehrungen/ST03_72pol_Zufuehrung, SFC *)
 PROGRAM ST03_72pol_Zufuehrung
VAR_OUTPUT
	SFCCurrentPOU		: STRING:='ST03_72pol_Zufuehrung';
	SFCCurrentStep		: STRING:='';
	FB_CurrentStepHistorie: FB_CurrentStepHistorie;
	SFCTime				: DINT;
	State   			: StateObject	:= STATE_WAIT;
	Result  			: StateResult;
END_VAR
VAR_INPUT
	Start				:BOOL;
END_VAR
VAR
	MsgOK				: BOOL;
	MsgCancel			: BOOL;
	SFCRun				: BOOL;
	SFCTimeStart		: TIME;
	Delay				: TON;
	(* Userdefinded area *)

END_VAR
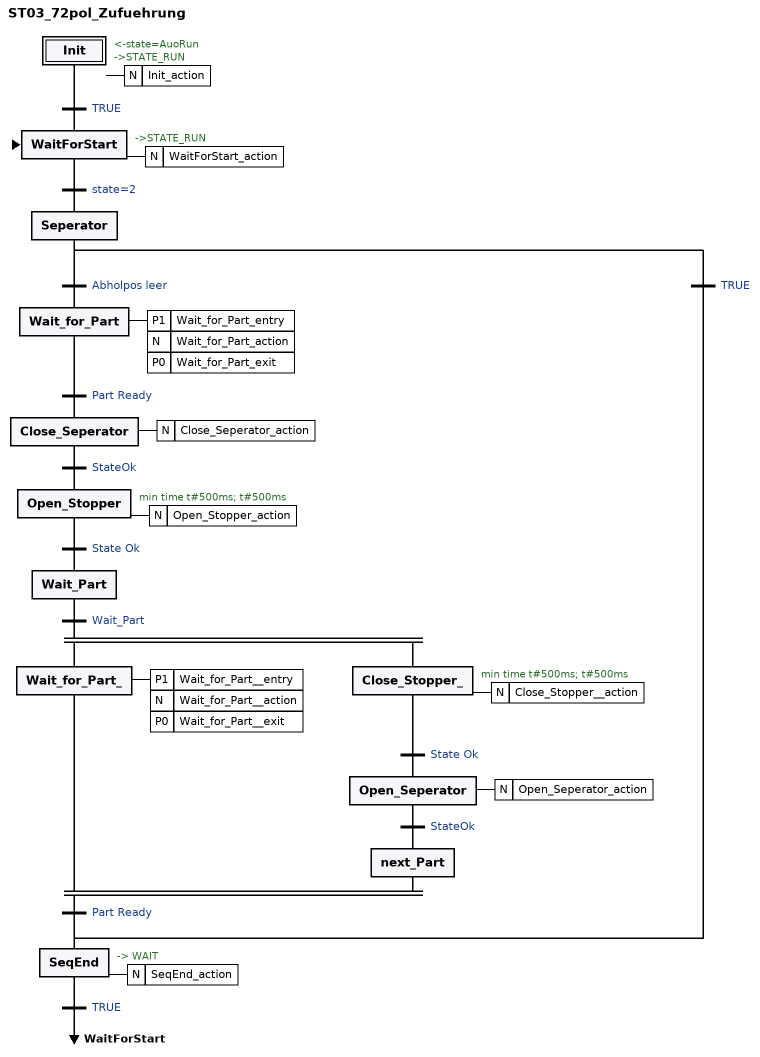
INITIAL_STEP Init: (* <-state=AuoRun / ->STATE_RUN *)
	Init_action(N);
END_STEP
TRANSITION FROM Init TO WaitForStart := TRUE;
END_TRANSITION
STEP WaitForStart: (* ->STATE_RUN *)
	WaitForStart_action(N);
END_STEP
TRANSITION FROM WaitForStart TO Seperator := state=2;
END_TRANSITION
STEP Seperator:
END_STEP
TRANSITION FROM Seperator TO Wait_for_Part := Abholpos leer;
END_TRANSITION
TRANSITION FROM Seperator TO SeqEnd := TRUE;
END_TRANSITION
STEP Wait_for_Part:
	Wait_for_Part_entry(P1);
	Wait_for_Part_action(N);
	Wait_for_Part_exit(P0);
END_STEP
TRANSITION FROM Wait_for_Part TO Close_Seperator := Part Ready;
END_TRANSITION
STEP Close_Seperator:
	Close_Seperator_action(N);
END_STEP
TRANSITION FROM Close_Seperator TO Open_Stopper := StateOk;
END_TRANSITION
STEP Open_Stopper: (* min time t#500ms; t#500ms *)
	Open_Stopper_action(N);
END_STEP
TRANSITION FROM Open_Stopper TO Wait_Part := State Ok;
END_TRANSITION
STEP Wait_Part:
END_STEP
TRANSITION FROM Wait_Part TO (Wait_for_Part_, Close_Stopper_) := Wait_Part;
END_TRANSITION
STEP Wait_for_Part_:
	Wait_for_Part__entry(P1);
	Wait_for_Part__action(N);
	Wait_for_Part__exit(P0);
END_STEP
STEP Close_Stopper_: (* min time t#500ms; t#500ms *)
	Close_Stopper__action(N);
END_STEP
TRANSITION FROM Close_Stopper_ TO Open_Seperator := State Ok;
END_TRANSITION
STEP Open_Seperator:
	Open_Seperator_action(N);
END_STEP
TRANSITION FROM Open_Seperator TO next_Part := StateOk;
END_TRANSITION
STEP next_Part:
END_STEP
TRANSITION FROM (Wait_for_Part_, next_Part) TO SeqEnd := Part Ready;
END_TRANSITION
STEP SeqEnd: (* -> WAIT *)
	SeqEnd_action(N);
END_STEP
TRANSITION FROM SeqEnd TO WaitForStart := TRUE;
END_TRANSITION

ACTION Init_action:
Start:=FALSE;
State:=STATE_WAIT;
MsgOK:=FALSE;
MsgCancel:=FALSE;
SFCRun:=FALSE;
Result:=RESULT_NON;
END_ACTION

ACTION WaitForStart_action:
IF 	Start   THEN
	State:=STATE_RUN;
	Result:=RESULT_NON;
	SFCTimeStart:=TIME();
	Start:=FALSE;
ELSE
	State:=STATE_WAIT;
	MsgOK:=FALSE;
	MsgCancel:=FALSE;
	SFCRun:=FALSE;
END_IF
END_ACTION

ACTION Wait_for_Part_entry:
ProcessMessage01:='';
Delay(IN:=FALSE);
END_ACTION

ACTION Wait_for_Part_action:
ProcessMessage01:='1IM9';(*warte auf Teil in Stopper*)
Delay(	IN:=ST03_546_B69_6.BitInToCheck,		(*  ISK an stopper.*)
		PT:=T#500ms);
END_ACTION

ACTION Wait_for_Part_exit:
ProcessMessage01:='';
Delay(IN:=FALSE);
END_ACTION

ACTION Close_Seperator_action:
ST03_547_Y70_1.MoveWork:=TRUE;		(*Zuführung Vereinzler AST/GST *)
END_ACTION

ACTION Open_Stopper_action:
ST03_547_Y70_2.MoveWork:=TRUE;		(* Züführung Stopper AST/GST *)
END_ACTION

ACTION Wait_for_Part__entry:
ProcessMessage01:='';
Delay(IN:=FALSE);
END_ACTION

ACTION Wait_for_Part__action:
ProcessMessage01:='1IM10';(*warte auf Teil in Abholposition*)
Delay(	IN:=	NOT ST03_Init_AbholPos.RoboPos31 AND
			NOT ST03_Init_AbholPos.RoboPos35,
		PT:=T#500ms);
END_ACTION

ACTION Wait_for_Part__exit:
ProcessMessage01:='';
Delay(IN:=FALSE);
END_ACTION

ACTION Close_Stopper__action:
ST03_547_Y70_2.MoveInit:=TRUE;		(* Züführung Stopper AST/GST *)
END_ACTION

ACTION Open_Seperator_action:
ST03_547_Y70_1.MoveInit:=TRUE;		(* Zuführung Vereinzler AST/GST *)
END_ACTION

ACTION SeqEnd_action:
SFCTime:=TIME_TO_DINT(TIME()-SFCTimeStart);
State:=STATE_WAIT;
END_ACTION

TRANSITION Abholpos leer:
NOT ST03_Init_AbholPos.RoboPos31 AND
NOT ST03_Init_AbholPos.RoboPos35
END_TRANSITION

TRANSITION Part Ready:
Delay.Q AND
NOT ST03_Init_AbholPos.RoboPos31 AND
NOT ST03_Init_AbholPos.RoboPos35 AND
ST03_546_B69_6.BitInToCheck	AND			(*ISK anwesend am Stoper*)
Robot01.ActualArea <> 4
END_TRANSITION

TRANSITION StateOk:
ST03_547_Y70_1.State=STATE_OK 	(* Zuführung Vereinzler AST/GST *)
END_TRANSITION

TRANSITION State Ok:
ST03_547_Y70_2.State=STATE_OK 	(* Züführung Stopper AST/GST *)
END_TRANSITION

TRANSITION Wait_Part:
ST03_Init_AbholPos.RoboPos31 OR
ST03_Init_AbholPos.RoboPos35
END_TRANSITION

TRANSITION State Ok:
ST03_547_Y70_2.State=STATE_OK 	(*Züführung Stopper AST/GST *)
END_TRANSITION

TRANSITION StateOk:
ST03_547_Y70_1.State=STATE_OK 	(* Zuführung Vereinzler AST/GST *)
END_TRANSITION

TRANSITION Part Ready:
Delay.Q AND
Robot01.ActualArea <> 4
END_TRANSITION
END_PROGRAM

(* POU Stations/ST_03_Ruestsaetze/ST_03_SFCs/Zufuehrungen/ST03_48pol_Zufuehrung, SFC *)
 PROGRAM ST03_48pol_Zufuehrung
VAR_OUTPUT
	SFCCurrentPOU		: STRING:='ST03_48pol_Zufuehrung';
	SFCCurrentStep		: STRING:='';
	FB_CurrentStepHistorie: FB_CurrentStepHistorie;
	SFCTime				: DINT;
	State   			: StateObject	:= STATE_WAIT;
	Result  			: StateResult;
END_VAR
VAR_INPUT
	Start				:BOOL;
END_VAR
VAR
	MsgOK				: BOOL;
	MsgCancel			: BOOL;
	SFCRun				: BOOL;
	SFCTimeStart		: TIME;
	Delay				: TON;
	(* Userdefinded area *)

END_VAR
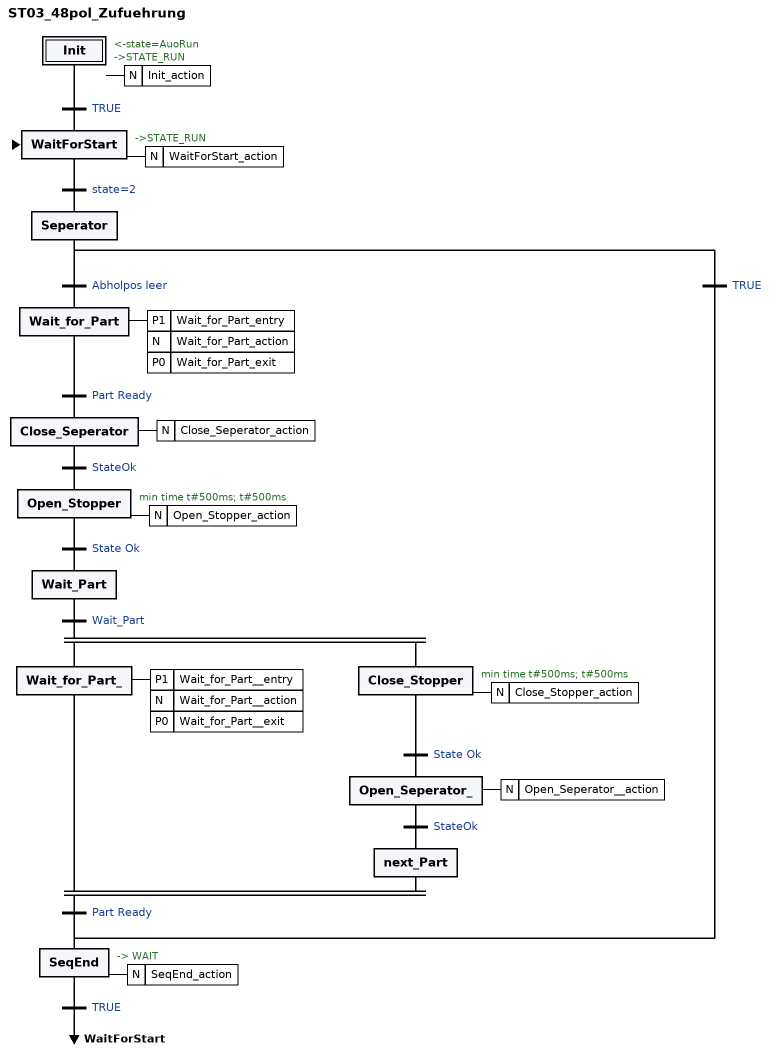
INITIAL_STEP Init: (* <-state=AuoRun / ->STATE_RUN *)
	Init_action(N);
END_STEP
TRANSITION FROM Init TO WaitForStart := TRUE;
END_TRANSITION
STEP WaitForStart: (* ->STATE_RUN *)
	WaitForStart_action(N);
END_STEP
TRANSITION FROM WaitForStart TO Seperator := state=2;
END_TRANSITION
STEP Seperator:
END_STEP
TRANSITION FROM Seperator TO Wait_for_Part := Abholpos leer;
END_TRANSITION
TRANSITION FROM Seperator TO SeqEnd := TRUE;
END_TRANSITION
STEP Wait_for_Part:
	Wait_for_Part_entry(P1);
	Wait_for_Part_action(N);
	Wait_for_Part_exit(P0);
END_STEP
TRANSITION FROM Wait_for_Part TO Close_Seperator := Part Ready;
END_TRANSITION
STEP Close_Seperator:
	Close_Seperator_action(N);
END_STEP
TRANSITION FROM Close_Seperator TO Open_Stopper := StateOk;
END_TRANSITION
STEP Open_Stopper: (* min time t#500ms; t#500ms *)
	Open_Stopper_action(N);
END_STEP
TRANSITION FROM Open_Stopper TO Wait_Part := State Ok;
END_TRANSITION
STEP Wait_Part:
END_STEP
TRANSITION FROM Wait_Part TO (Wait_for_Part_, Close_Stopper) := Wait_Part;
END_TRANSITION
STEP Wait_for_Part_:
	Wait_for_Part__entry(P1);
	Wait_for_Part__action(N);
	Wait_for_Part__exit(P0);
END_STEP
STEP Close_Stopper: (* min time t#500ms; t#500ms *)
	Close_Stopper_action(N);
END_STEP
TRANSITION FROM Close_Stopper TO Open_Seperator_ := State Ok;
END_TRANSITION
STEP Open_Seperator_:
	Open_Seperator__action(N);
END_STEP
TRANSITION FROM Open_Seperator_ TO next_Part := StateOk;
END_TRANSITION
STEP next_Part:
END_STEP
TRANSITION FROM (Wait_for_Part_, next_Part) TO SeqEnd := Part Ready;
END_TRANSITION
STEP SeqEnd: (* -> WAIT *)
	SeqEnd_action(N);
END_STEP
TRANSITION FROM SeqEnd TO WaitForStart := TRUE;
END_TRANSITION

ACTION Init_action:
Start:=FALSE;
State:=STATE_WAIT;
MsgOK:=FALSE;
MsgCancel:=FALSE;
SFCRun:=FALSE;
Result:=RESULT_NON;
END_ACTION

ACTION WaitForStart_action:
IF 	Start   THEN
	State:=STATE_RUN;
	Result:=RESULT_NON;
	SFCTimeStart:=TIME();
	Start:=FALSE;
ELSE
	State:=STATE_WAIT;
	MsgOK:=FALSE;
	MsgCancel:=FALSE;
	SFCRun:=FALSE;
END_IF
END_ACTION

ACTION Wait_for_Part_entry:
ProcessMessage01:='';
Delay(IN:=FALSE);
END_ACTION

ACTION Wait_for_Part_action:
ProcessMessage01:='1IM9';(*warte auf Teil in Stopper*)
Delay(	IN:=ST03_551_B69_6.BitInToCheck, 		(*  ISK an stopper.*)
		PT:=T#500ms);
END_ACTION

ACTION Wait_for_Part_exit:
ProcessMessage01:='';
Delay(IN:=FALSE);
END_ACTION

ACTION Close_Seperator_action:
ST03_552_Y70_1.MoveWork:=TRUE;		(*Zuführung Vereinzler AST/GST *)
END_ACTION

ACTION Open_Stopper_action:
ST03_552_Y70_2.MoveWork:=TRUE;		(* Züführung Stopper AST/GST *)
END_ACTION

ACTION Wait_for_Part__entry:
ProcessMessage01:='';
Delay(IN:=FALSE);
END_ACTION

ACTION Wait_for_Part__action:
ProcessMessage01:='1IM10';(*warte auf Teil in Abholposition*)
Delay(	IN:=	NOT ST03_Init_AbholPos.RoboPos31 AND
			NOT ST03_Init_AbholPos.RoboPos35,
		PT:=T#500ms);
END_ACTION

ACTION Wait_for_Part__exit:
ProcessMessage01:='';
Delay(IN:=FALSE);
END_ACTION

ACTION Close_Stopper_action:
ST03_552_Y70_2.MoveInit:=TRUE;		(* Züführung Stopper AST/GST *)
END_ACTION

ACTION Open_Seperator__action:
ST03_552_Y70_1.MoveInit:=TRUE;		(*Zuführung Vereinzler AST/GST *)
END_ACTION

ACTION SeqEnd_action:
SFCTime:=TIME_TO_DINT(TIME()-SFCTimeStart);
State:=STATE_WAIT;
END_ACTION

TRANSITION Abholpos leer:
NOT ST03_Init_AbholPos.RoboPos31 AND
NOT ST03_Init_AbholPos.RoboPos35
END_TRANSITION

TRANSITION Part Ready:
Delay.Q AND
NOT ST03_Init_AbholPos.RoboPos31 AND
NOT ST03_Init_AbholPos.RoboPos35 AND
ST03_551_B69_6.BitInToCheck	AND			(*ISK anwesend am Stoper*)
Robot01.ActualArea <> 4
END_TRANSITION

TRANSITION StateOk:
ST03_552_Y70_1.State=STATE_OK 	(* Zuführung Vereinzler AST/GST *)
END_TRANSITION

TRANSITION State Ok:
ST03_552_Y70_2.State=STATE_OK 	(* Züführung Stopper AST/GST *)
END_TRANSITION

TRANSITION Wait_Part:
ST03_Init_AbholPos.RoboPos31 OR
ST03_Init_AbholPos.RoboPos35
END_TRANSITION

TRANSITION State Ok:
ST03_552_Y70_2.State=STATE_OK 	(*Züführung Stopper AST/GST *)
END_TRANSITION

TRANSITION StateOk:
ST03_552_Y70_1.State=STATE_OK 	(* Zuführung Vereinzler AST/GST *)
END_TRANSITION

TRANSITION Part Ready:
Delay.Q AND
Robot01.ActualArea <> 4
END_TRANSITION
END_PROGRAM

(* POU Stations/ST_03_Ruestsaetze/ST_03_SFCs/Zufuehrungen/ST03_268pol_Zufuehrung, SFC *)
PROGRAM ST03_268pol_Zufuehrung
VAR_INPUT
	Start					:BOOL;
END_VAR
VAR_OUTPUT
	SFCCurrentPOU			: STRING:='ST03_268pol_Zufuehrung';
	SFCCurrentStep			: STRING:='';
	FB_CurrentStepHistorie: FB_CurrentStepHistorie;
	SFCTime				: DINT;
	State   					: StateObject	:= STATE_WAIT;
	Result  					: ARRAY [1..NO_OF_RESULT] OF StateResult;
	ResultOK				: BOOL;
END_VAR
VAR
	MsgOK				: BOOL;
	MsgCancel			: BOOL;
	SFCRun			: BOOL;
	SFCTimeStart		: TIME;
	Delay				: TON;
	(* Userdefinded area *)

	i					: INT;
	Pos					: INT;
	RepeatCounter		: INT;
	NokCounter			: INT;
	NokCounterPercent	: INT;
  	NokPercent   		: ARRAY[1..100] OF BOOL;
	CamAlwaysOK		:BOOL:=TRUE;		(*schreibt immer OK nur zum Testen*)

END_VAR

VAR CONSTANT
	NO_OF_RESULT	: INT :=2;
END_VAR
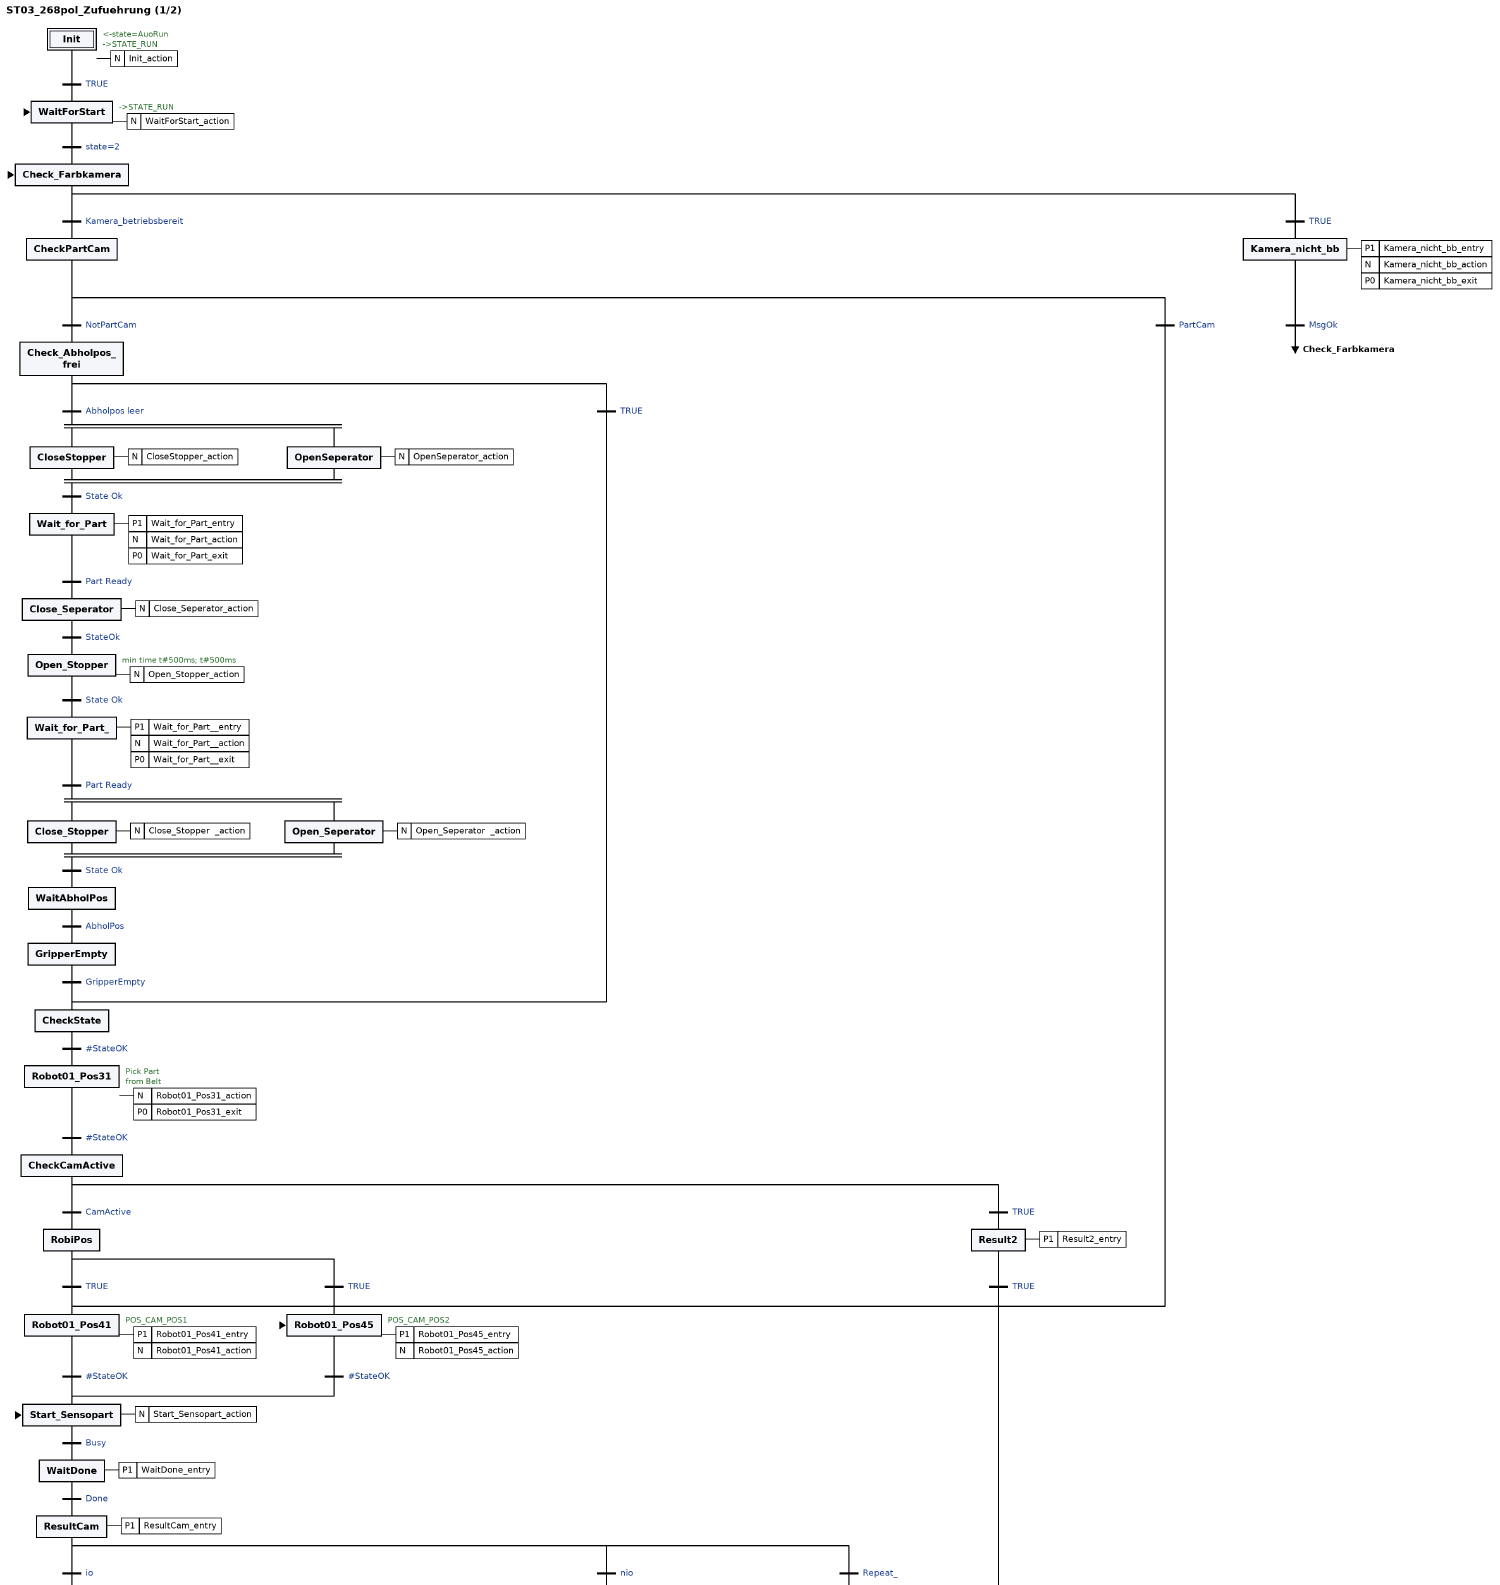
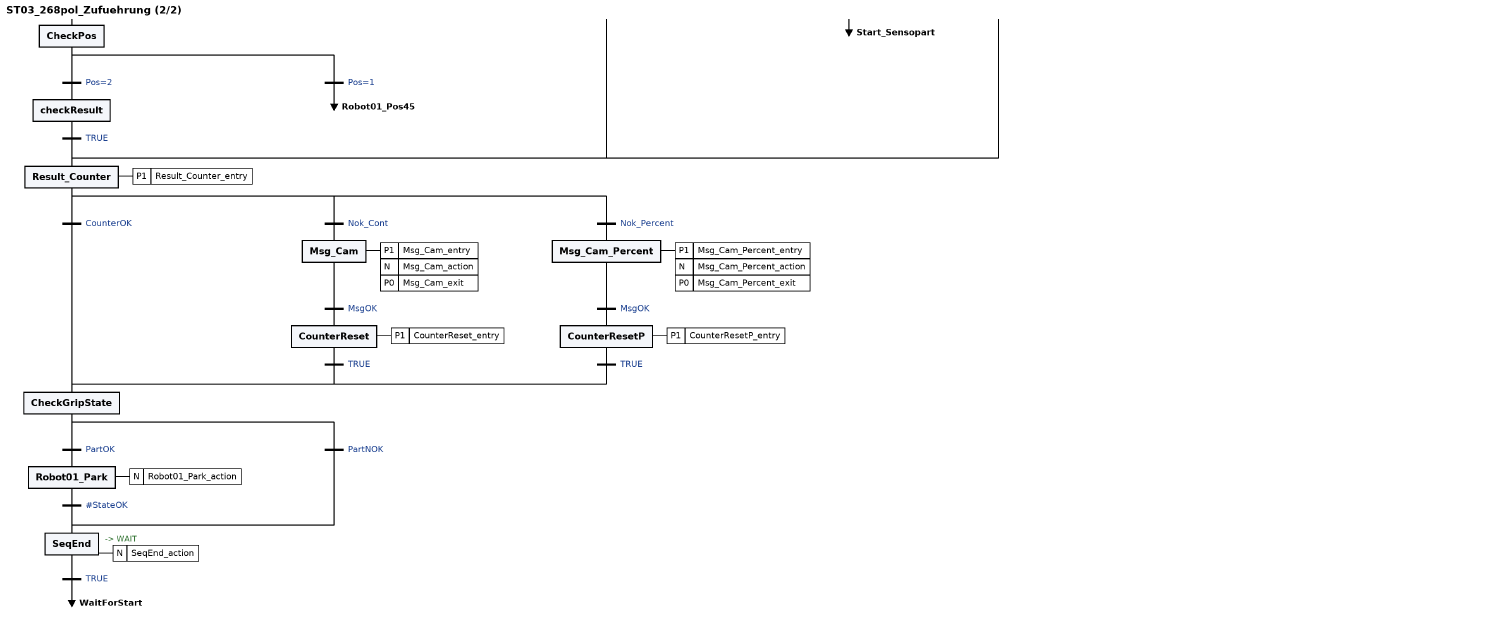
INITIAL_STEP Init: (* <-state=AuoRun / ->STATE_RUN *)
	Init_action(N);
END_STEP
TRANSITION FROM Init TO WaitForStart := TRUE;
END_TRANSITION
STEP WaitForStart: (* ->STATE_RUN *)
	WaitForStart_action(N);
END_STEP
TRANSITION FROM WaitForStart TO Check_Farbkamera := state=2;
END_TRANSITION
STEP Check_Farbkamera:
END_STEP
TRANSITION FROM Check_Farbkamera TO CheckPartCam := Kamera_betriebsbereit;
END_TRANSITION
TRANSITION FROM Check_Farbkamera TO Kamera_nicht_bb := TRUE;
END_TRANSITION
STEP CheckPartCam:
END_STEP
TRANSITION FROM CheckPartCam TO Check_Abholpos_frei := NotPartCam;
END_TRANSITION
TRANSITION FROM CheckPartCam TO Robot01_Pos41 := PartCam;
END_TRANSITION
STEP Check_Abholpos_frei:
END_STEP
TRANSITION FROM Check_Abholpos_frei TO (CloseStopper, OpenSeperator) := Abholpos leer;
END_TRANSITION
TRANSITION FROM Check_Abholpos_frei TO CheckState := TRUE;
END_TRANSITION
STEP CloseStopper:
	CloseStopper_action(N);
END_STEP
STEP OpenSeperator:
	OpenSeperator_action(N);
END_STEP
TRANSITION FROM (CloseStopper, OpenSeperator) TO Wait_for_Part := State Ok;
END_TRANSITION
STEP Kamera_nicht_bb:
	Kamera_nicht_bb_entry(P1);
	Kamera_nicht_bb_action(N);
	Kamera_nicht_bb_exit(P0);
END_STEP
TRANSITION FROM Kamera_nicht_bb TO Check_Farbkamera := MsgOk;
END_TRANSITION
STEP Wait_for_Part:
	Wait_for_Part_entry(P1);
	Wait_for_Part_action(N);
	Wait_for_Part_exit(P0);
END_STEP
TRANSITION FROM Wait_for_Part TO Close_Seperator := Part Ready;
END_TRANSITION
STEP Close_Seperator:
	Close_Seperator_action(N);
END_STEP
TRANSITION FROM Close_Seperator TO Open_Stopper := StateOk;
END_TRANSITION
STEP Open_Stopper: (* min time t#500ms; t#500ms *)
	Open_Stopper_action(N);
END_STEP
TRANSITION FROM Open_Stopper TO Wait_for_Part_ := State Ok;
END_TRANSITION
STEP Wait_for_Part_:
	Wait_for_Part__entry(P1);
	Wait_for_Part__action(N);
	Wait_for_Part__exit(P0);
END_STEP
TRANSITION FROM Wait_for_Part_ TO (Close_Stopper  , Open_Seperator  ) := Part Ready;
END_TRANSITION
STEP Close_Stopper  :
	Close_Stopper  _action(N);
END_STEP
STEP Open_Seperator  :
	Open_Seperator  _action(N);
END_STEP
TRANSITION FROM (Close_Stopper  , Open_Seperator  ) TO WaitAbholPos := State Ok;
END_TRANSITION
STEP WaitAbholPos:
END_STEP
TRANSITION FROM WaitAbholPos TO GripperEmpty := AbholPos;
END_TRANSITION
STEP GripperEmpty:
END_STEP
TRANSITION FROM GripperEmpty TO CheckState := GripperEmpty;
END_TRANSITION
STEP CheckState:
END_STEP
TRANSITION FROM CheckState TO Robot01_Pos31 := #StateOK;
END_TRANSITION
STEP Robot01_Pos31: (* Pick Part / from Belt *)
	Robot01_Pos31_action(N);
	Robot01_Pos31_exit(P0);
END_STEP
TRANSITION FROM Robot01_Pos31 TO CheckCamActive := #StateOK;
END_TRANSITION
STEP CheckCamActive:
END_STEP
TRANSITION FROM CheckCamActive TO RobiPos := CamActive;
END_TRANSITION
TRANSITION FROM CheckCamActive TO Result2 := TRUE;
END_TRANSITION
STEP RobiPos:
END_STEP
TRANSITION FROM RobiPos TO Robot01_Pos41 := TRUE;
END_TRANSITION
TRANSITION FROM RobiPos TO Robot01_Pos45 := TRUE;
END_TRANSITION
STEP Robot01_Pos41: (* POS_CAM_POS1 *)
	Robot01_Pos41_entry(P1);
	Robot01_Pos41_action(N);
END_STEP
TRANSITION FROM Robot01_Pos41 TO Start_Sensopart := #StateOK;
END_TRANSITION
STEP Robot01_Pos45: (* POS_CAM_POS2 *)
	Robot01_Pos45_entry(P1);
	Robot01_Pos45_action(N);
END_STEP
TRANSITION FROM Robot01_Pos45 TO Start_Sensopart := #StateOK;
END_TRANSITION
STEP Start_Sensopart:
	Start_Sensopart_action(N);
END_STEP
TRANSITION FROM Start_Sensopart TO WaitDone := Busy;
END_TRANSITION
STEP WaitDone:
	WaitDone_entry(P1);
END_STEP
TRANSITION FROM WaitDone TO ResultCam := Done;
END_TRANSITION
STEP ResultCam:
	ResultCam_entry(P1);
END_STEP
TRANSITION FROM ResultCam TO CheckPos := io;
END_TRANSITION
TRANSITION FROM ResultCam TO Result_Counter := nio;
END_TRANSITION
TRANSITION FROM ResultCam TO Start_Sensopart := Repeat_;
END_TRANSITION
STEP CheckPos:
END_STEP
TRANSITION FROM CheckPos TO checkResult := Pos=2;
END_TRANSITION
TRANSITION FROM CheckPos TO Robot01_Pos45 := Pos=1;
END_TRANSITION
STEP checkResult:
END_STEP
TRANSITION FROM checkResult TO Result_Counter := TRUE;
END_TRANSITION
STEP Result2:
	Result2_entry(P1);
END_STEP
TRANSITION FROM Result2 TO Result_Counter := TRUE;
END_TRANSITION
STEP Result_Counter:
	Result_Counter_entry(P1);
END_STEP
TRANSITION FROM Result_Counter TO CheckGripState := CounterOK;
END_TRANSITION
TRANSITION FROM Result_Counter TO Msg_Cam := Nok_Cont;
END_TRANSITION
TRANSITION FROM Result_Counter TO Msg_Cam_Percent := Nok_Percent;
END_TRANSITION
STEP Msg_Cam:
	Msg_Cam_entry(P1);
	Msg_Cam_action(N);
	Msg_Cam_exit(P0);
END_STEP
TRANSITION FROM Msg_Cam TO CounterReset := MsgOK;
END_TRANSITION
STEP CounterReset:
	CounterReset_entry(P1);
END_STEP
TRANSITION FROM CounterReset TO CheckGripState := TRUE;
END_TRANSITION
STEP Msg_Cam_Percent:
	Msg_Cam_Percent_entry(P1);
	Msg_Cam_Percent_action(N);
	Msg_Cam_Percent_exit(P0);
END_STEP
TRANSITION FROM Msg_Cam_Percent TO CounterResetP := MsgOK;
END_TRANSITION
STEP CounterResetP:
	CounterResetP_entry(P1);
END_STEP
TRANSITION FROM CounterResetP TO CheckGripState := TRUE;
END_TRANSITION
STEP CheckGripState:
END_STEP
TRANSITION FROM CheckGripState TO Robot01_Park := PartOK;
END_TRANSITION
TRANSITION FROM CheckGripState TO SeqEnd := PartNOK;
END_TRANSITION
STEP Robot01_Park:
	Robot01_Park_action(N);
END_STEP
TRANSITION FROM Robot01_Park TO SeqEnd := #StateOK;
END_TRANSITION
STEP SeqEnd: (* -> WAIT *)
	SeqEnd_action(N);
END_STEP
TRANSITION FROM SeqEnd TO WaitForStart := TRUE;
END_TRANSITION

ACTION Init_action:
Start:=FALSE;
State:=STATE_WAIT;
MsgOK:=FALSE;
MsgCancel:=FALSE;
SFCRun:=FALSE;
NokCounter:=0;
i:=1;
Pos:=1;
FOR i:=1 TO NO_OF_RESULT BY 1 DO
	Result[i]:=RESULT_NON;
END_FOR;
END_ACTION

ACTION WaitForStart_action:
i:=1;
IF 	Start   THEN
	State:=STATE_RUN;
	SFCTimeStart:=TIME();
	Start:=FALSE;
	FOR i:=1 TO NO_OF_RESULT BY 1 DO
		Result[i]:=RESULT_NON;
	END_FOR
	Pos:=1;
ELSE
	State:=STATE_WAIT;
	MsgOK:=FALSE;
	MsgCancel:=FALSE;
	SFCRun:=FALSE;
END_IF
END_ACTION

ACTION CloseStopper_action:
ST03_557_Y70_2.MoveInit:=TRUE;		(* Züführung Stopper AST/GST *)
END_ACTION

ACTION OpenSeperator_action:
ST03_557_Y70_1.MoveInit:=TRUE;		(* Zuführung Vereinzler AST/GST *)
END_ACTION

ACTION Kamera_nicht_bb_entry:
MessageHandler.ClearMessageLines(sVisu:=Visu.Message);
END_ACTION

ACTION Kamera_nicht_bb_action:
MessageHandler.Msg.ID:='PM152';
MessageHandler.Msg.Name:='Check Camera';
MessageHandler.Msg.Text:='Sesopart Kamera ist nicht betriebsbereit';
MessageHandler.Msg.Color:=Color.red;
MessageHandler.Msg.Station:=1;


MessageHandler(
	Prio:=2, 							(*1=highest, .. , 4=lowest*)
	Btn1Addr:=ADR(MsgOk),			(*Address of Button1 , if Zero then Button is unvisible*)
	Btn2Addr:=,						(*Address of Button2 , if Zero then Button is unvisible*)
	sVisu:=Visu.Message);
END_ACTION

ACTION Kamera_nicht_bb_exit:
MsgOk:=FALSE;
MsgCancel:=FALSE;
ST02_DT_95_A1.b_quitt:=TRUE;
END_ACTION

ACTION Wait_for_Part_entry:
ProcessMessage01:='';
Delay.IN:=FALSE;
Delay();
END_ACTION

ACTION Wait_for_Part_action:
ProcessMessage01:='1IM9';(*warte auf Teil in Stopper*)
Delay.IN:=ST03_556_B69_6.BitInToCheck; 		(*  ISK an Stopper.*)
Delay.PT:=T#500ms;
Delay();
END_ACTION

ACTION Wait_for_Part_exit:
ProcessMessage01:='';
END_ACTION

ACTION Close_Seperator_action:
ST03_557_Y70_1.MoveWork:=TRUE;		(*Zuführung Vereinzler AST/GST *)
END_ACTION

ACTION Open_Stopper_action:
ST03_557_Y70_2.MoveWork:=TRUE;		(* Züführung Stopper AST/GST *)
END_ACTION

ACTION Wait_for_Part__entry:
ProcessMessage01:='';
Delay(IN:=FALSE);
END_ACTION

ACTION Wait_for_Part__action:
ProcessMessage01:='1IM10';(*warte auf Teil in Abholposition*)
Delay(	IN:=	ST03_Init_AbholPos.RoboPos31,
		PT:=T#500ms);
END_ACTION

ACTION Wait_for_Part__exit:
ProcessMessage01:='';
Delay(IN:=FALSE);
END_ACTION

ACTION Close_Stopper  _action:
ST03_557_Y70_2.MoveInit:=TRUE;		(* Züführung Stopper AST/GST *)
END_ACTION

ACTION Open_Seperator  _action:
ST03_557_Y70_1.MoveInit:=TRUE;		(* Zuführung Vereinzler AST/GST *)
END_ACTION

ACTION Robot01_Pos31_action:
Robot01.PosNo:=POS_WT_POS1;
Robot01.PosOffset:=gRobotOffset;
Robot01.Override:=MP.ST00.Override;
Robot01.SetToolOn:=FALSE;
Robot01.SetToolOff:=TRUE;
Robot01.ExecuteMove:=TRUE;
END_ACTION

ACTION Robot01_Pos31_exit:
gRob01GripState:=PART_CAM;
FOR i:=1 TO NO_OF_RESULT BY 1 DO
	Result[i]:=0;
END_FOR
END_ACTION

ACTION Robot01_Pos41_entry:
RepeatCounter:=0;
END_ACTION

ACTION Robot01_Pos41_action:
Robot01.PosNo:=POS_CAM_POS1;
Robot01.PosOffset:=gRobotOffset;
Robot01.Override:=MP.ST00.Override;
Robot01.SetToolOn:=FALSE;
Robot01.SetToolOff:=TRUE;
Robot01.ExecuteMove:=TRUE;
Pos:=1;
END_ACTION

ACTION Robot01_Pos45_entry:
RepeatCounter:=0;
END_ACTION

ACTION Robot01_Pos45_action:
Robot01.PosNo:=POS_CAM_POS2;
Robot01.PosOffset:=gRobotOffset;
Robot01.Override:=MP.ST00.Override;
Robot01.SetToolOn:=FALSE;
Robot01.SetToolOff:=TRUE;
Robot01.ExecuteMove:=TRUE;
Pos:=2;
END_ACTION

ACTION Start_Sensopart_action:
ST03_8_100_A1.JobNo := TD.Sensopart_CamProgNo ;
ST03_8_100_A1.st_ctrl_in.b_start := TRUE;
END_ACTION

ACTION WaitDone_entry:
ST03_8_100_A1.st_ctrl_in.b_start := FALSE;
RepeatCounter:=RepeatCounter+1;
END_ACTION

ACTION ResultCam_entry:
IF 	(ST03_8_100_A1.b_Kam_Pruef_IO AND	 (*Kamera Farberkennung*)
	NOT ST03_8_100_A1.b_Kam_Pruef_NIO) THEN
	Result[Pos]:=RESULT_OK;
ELSE
	Result[Pos]:=RESULT_NOK;
END_IF
END_ACTION

ACTION Result2_entry:
FOR i:=1 TO NO_OF_RESULT BY 1 DO
	Result[i]:=RESULT_OK;
END_FOR
END_ACTION

ACTION Result_Counter_entry:
FOR i:=100 TO 2 BY-1 DO
   	NokPercent[i] := NokPercent[i-1];
END_FOR

ResultOk:=TRUE;
FOR i:=1 TO NO_OF_RESULT BY 1 DO
	IF	ResultOk AND Result[i] = RESULT_NOK 	THEN
		ResultOk:=FALSE;
	END_IF
END_FOR

IF 	ResultOk OR
	CamAlwaysOK THEN		(*schreibt immer NOK nur zum Testen*)
	NokCounter:=0;
	NokPercent[1] := FALSE;
	gRob01GripState:=PART_OK;
ELSE
	NokCounter:=NokCounter+1;
	NokPercent[1] := TRUE;
	gRob01GripState:=PART_NOK;
END_IF
END_ACTION

ACTION Msg_Cam_entry:
MessageHandler.ClearMessageLines(sVisu:=Visu.Message);
END_ACTION

ACTION Msg_Cam_action:
MessageHandler.Msg.ID:='PM112';
MessageHandler.Msg.Name:='Sensopart Kam.-Erg. Prüfung  n.i.o:';
MessageHandler.Msg.Text:='Sensopart Kam.-Erg. Prüfung  n.i.o: Fehler in Folge';
MessageHandler.Msg.Color:=Color.red;
MessageHandler.Msg.Station:=3;
MessageHandler.MsgButton1Text:='continue';

MessageHandler(
	Prio:=2, 								(*1=highest, .. , 4=lowest*)
	Btn1Addr:=ADR(MsgOk),				(*Address of Button1 , if Zero then Button is unvisible*)
	Btn2Addr:=0(*ADR(MsgCancel)*),			(*Address of Button2 , if Zero then Button is unvisible*)
	sVisu:=Visu.Message);
END_ACTION

ACTION Msg_Cam_exit:
MsgOk:=FALSE;
MsgCancel:=FALSE;
END_ACTION

ACTION CounterReset_entry:
NokCounter:=0;
END_ACTION

ACTION Msg_Cam_Percent_entry:
MessageHandler.ClearMessageLines(sVisu:=Visu.Message);
END_ACTION

ACTION Msg_Cam_Percent_action:
MessageHandler.Msg.ID:='PM113';
MessageHandler.Msg.Name:='Sensopart Kam.-Erg. Prüfung  n.i.o:';
MessageHandler.Msg.Text:='Sensopart Kam.-Erg. Prüfung  n.i.o:% Fehler';
MessageHandler.Msg.Color:=Color.red;
MessageHandler.Msg.Station:=3;
MessageHandler.MsgButton1Text:='continue';

MessageHandler(
	Prio:=2, 								(*1=highest, .. , 4=lowest*)
	Btn1Addr:=ADR(MsgOk),				(*Address of Button1 , if Zero then Button is unvisible*)
	Btn2Addr:=0(*ADR(MsgCancel)*),			(*Address of Button2 , if Zero then Button is unvisible*)
	sVisu:=Visu.Message);
END_ACTION

ACTION Msg_Cam_Percent_exit:
MsgOk:=FALSE;
MsgCancel:=FALSE;
END_ACTION

ACTION CounterResetP_entry:
NokCounter:=0;
(*Percent Register löschen*)
FOR i:=1 TO 100 BY 1 DO
  NokPercent[i]:= FALSE;
END_FOR
END_ACTION

ACTION Robot01_Park_action:
Robot01.PosNo:=POS_PARK;
Robot01.PosOffset:=gRobotOffset;
Robot01.Override:=MP.ST00.Override;
Robot01.SetToolOn:=FALSE;
Robot01.SetToolOff:=TRUE;
Robot01.ExecuteMove:=TRUE;
END_ACTION

ACTION SeqEnd_action:
SFCTime:=TIME_TO_DINT(TIME()-SFCTimeStart);
State:=STATE_WAIT;
END_ACTION

TRANSITION Kamera_betriebsbereit:
(*Kamera Farberkennung*)
(
NOT ST03_8_100_A1.sm_kamera_nicht_bb OR
NOT ST03_8_100_A1.Activated	)
END_TRANSITION

TRANSITION NotPartCam:
gRob01GripState<>PART_CAM
END_TRANSITION

TRANSITION Abholpos leer:
NOT ST03_Init_AbholPos.RoboPos31
END_TRANSITION

TRANSITION PartCam:
TRUE
END_TRANSITION

TRANSITION State Ok:
ST03_557_Y70_2.State=STATE_OK AND	(*Züführung Stopper AST/GST *)
ST03_557_Y70_1.State=STATE_OK			(* Zuführung Vereinzler AST/GST *)
END_TRANSITION

TRANSITION Part Ready:
Delay.Q AND
NOT ST03_Init_AbholPos.RoboPos31 AND
ST03_556_B69_6.BitInToCheck	AND			(*ISK anwesend am Stoper*)
Robot01.ActualArea <> 4
END_TRANSITION

TRANSITION StateOk:
ST03_557_Y70_1.State=STATE_OK AND	(* Zuführung Vereinzler AST/GST *)
Robot01.ActualArea <> 3 AND
Robot01.ActualArea <> 4
END_TRANSITION

TRANSITION State Ok:
ST03_557_Y70_2.State=STATE_OK 	(* Züführung Stopper AST/GST *)
END_TRANSITION

TRANSITION Part Ready:
Delay.Q AND
Robot01.ActualArea <> 4
END_TRANSITION

TRANSITION State Ok:
ST03_557_Y70_2.State=STATE_OK AND	(*Züführung Stopper AST/GST *)
ST03_557_Y70_1.State=STATE_OK			(* Zuführung Vereinzler AST/GST *)
END_TRANSITION

TRANSITION AbholPos:
ST03_556_B69_7. BitInToCheck (*ISK anwesend an Abholposition*)
END_TRANSITION

TRANSITION GripperEmpty:
gRob01GripState=PART_NO AND
Robot01.RemInToolWorkSensor
END_TRANSITION

TRANSITION #StateOK:
Robot01.State=STATE_WAIT AND
gRob01GripState=PART_NO
END_TRANSITION

TRANSITION #StateOK:
Robot01.State=STATE_OK AND
gTipImp
END_TRANSITION

TRANSITION CamActive:
ST03_8_100_A1.Activated
END_TRANSITION

TRANSITION #StateOK:
Robot01.State=STATE_OK AND
gTipImp
END_TRANSITION

TRANSITION #StateOK:
Robot01.State=STATE_OK AND
gTipImp
END_TRANSITION

TRANSITION Busy:
ST03_8_100_A1.st_ctrl_out.b_busy (*Kamera Farberkennung Ehternet*)
END_TRANSITION

TRANSITION Done:
ST03_8_100_A1.st_ctrl_out.b_fertig
END_TRANSITION

TRANSITION io:
Result[Pos]=RESULT_OK
END_TRANSITION

TRANSITION nio:
RepeatCounter>=2
END_TRANSITION

TRANSITION Repeat_:
TRUE
END_TRANSITION

TRANSITION CounterOK:
(NokCounter<MP.ST03.CamNoOfErrors AND
NokCounterPercent < MP.ST02.CamNoOfErrorsPercent) OR
CamAlwaysOk
END_TRANSITION

TRANSITION Nok_Cont:
NokCounter >= MP.ST03.CamNoOfErrors
END_TRANSITION

TRANSITION Nok_Percent:
NokCounterPercent >= MP.ST03.CamNoOfErrorsPercent
END_TRANSITION

TRANSITION PartOK:
gRob01GripState=PART_OK
END_TRANSITION

TRANSITION #StateOK:
Robot01.State=STATE_OK AND
gTipImp
END_TRANSITION

TRANSITION PartNOK:
(*NIO Pos wird im ST03_Main angefahren*)
gRob01GripState=PART_NOK
END_TRANSITION
END_PROGRAM

(* POU Stations/ST_03_Ruestsaetze/ST_03_SFCs/Zufuehrungen/ST03_102pol_neu_Zufuehrung, SFC *)
PROGRAM ST03_102pol_neu_Zufuehrung
VAR_INPUT
	Start					:BOOL;
END_VAR
VAR_OUTPUT
	SFCCurrentPOU			: STRING:='ST03_102pol_neu_Zufuehrung';
	SFCCurrentStep			: STRING:='';
	FB_CurrentStepHistorie	: FB_CurrentStepHistorie;
	SFCTime				: DINT;
	State   					: StateObject	:= STATE_WAIT;
	ResultCam				: ARRAY [1..NO_OF_RESULT] OF StateResult;
	ResultOK				: BOOL;
END_VAR
VAR
	MsgOK				: BOOL;
	MsgCancel			: BOOL;
	SFCRun			: BOOL;
	SFCTimeStart		: TIME;
	Delay				: TON;
	(* Userdefinded area *)

	i					: INT:=1;
	Pos					: INT:= 1;
	RepeatCounter		: INT;
	NokCounter			: INT;
	NokCounterPercent	: INT;
  	NokPercent   		: ARRAY[1..100] OF BOOL;
	CamAlwaysOK		: ARRAY[1..2] OF BOOL:=TRUE,TRUE;		(*schreibt immer OK nur zum Testen*)
END_VAR

VAR CONSTANT
	NO_OF_RESULT	: INT :=4;
END_VAR
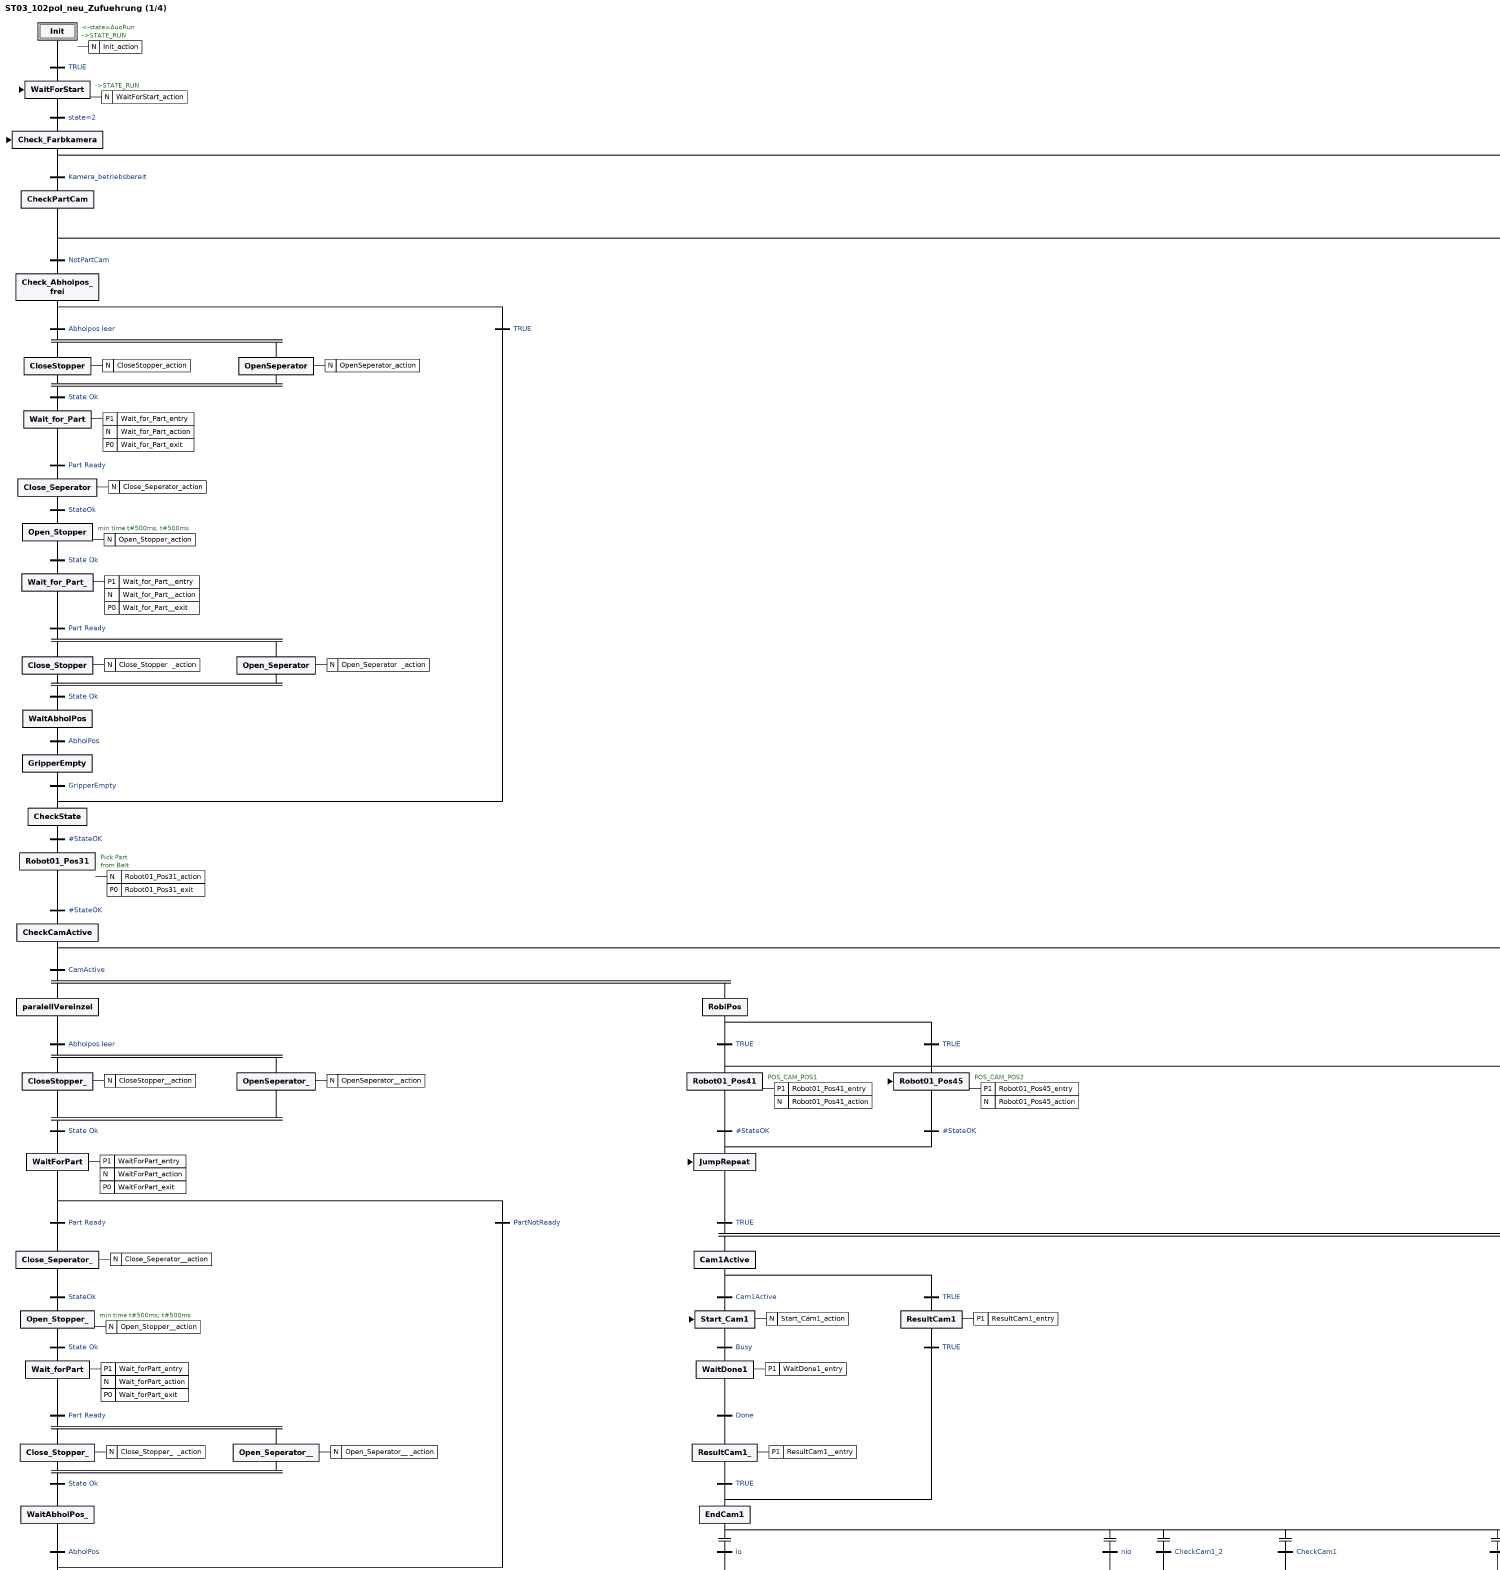
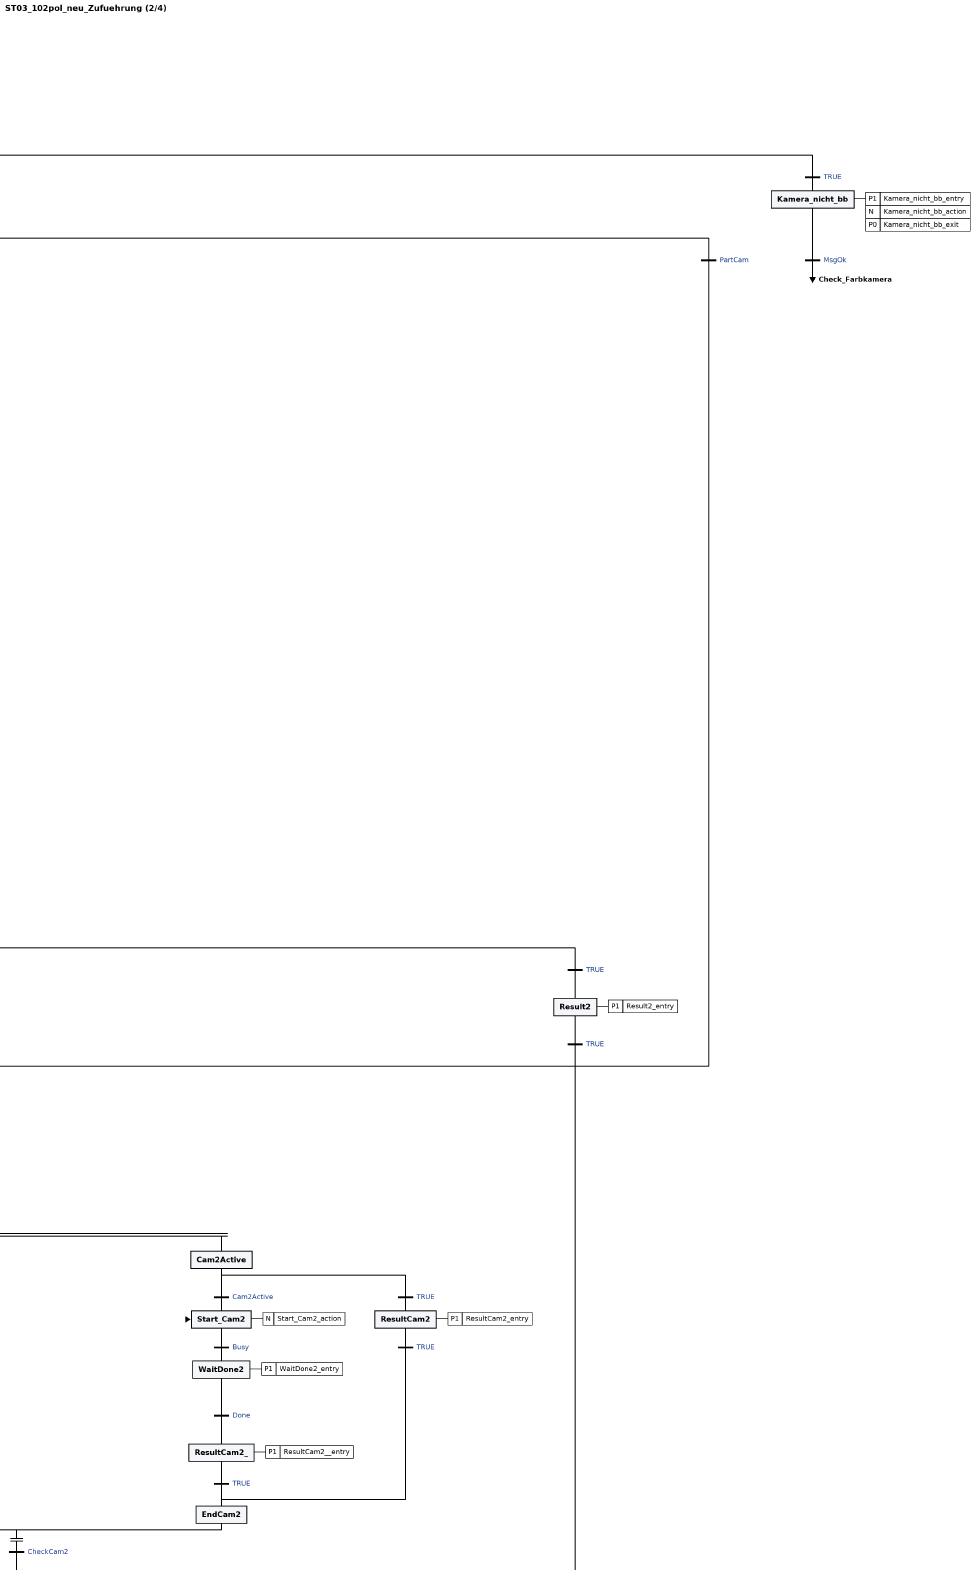
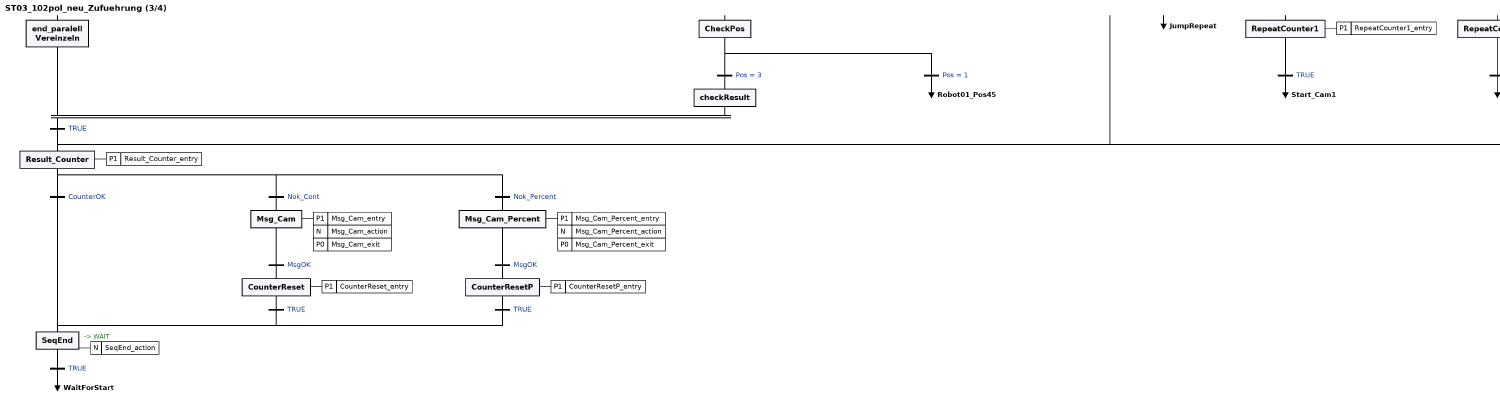
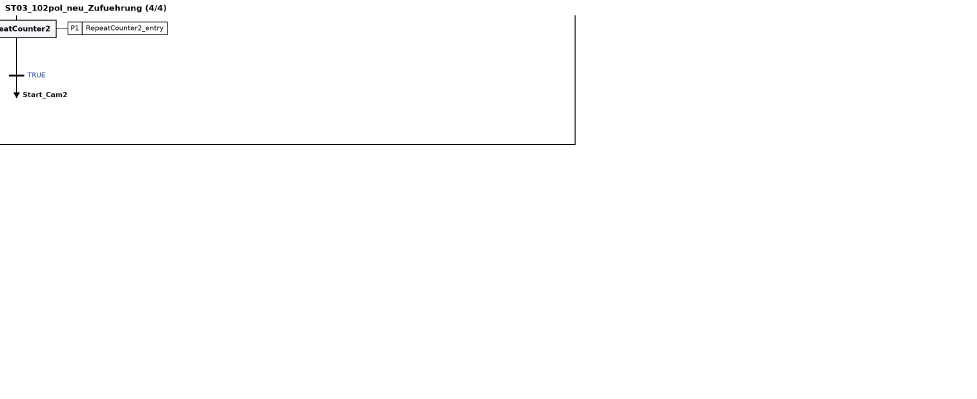
INITIAL_STEP Init: (* <-state=AuoRun / ->STATE_RUN *)
	Init_action(N);
END_STEP
TRANSITION FROM Init TO WaitForStart := TRUE;
END_TRANSITION
STEP WaitForStart: (* ->STATE_RUN *)
	WaitForStart_action(N);
END_STEP
TRANSITION FROM WaitForStart TO Check_Farbkamera := state=2;
END_TRANSITION
STEP Check_Farbkamera:
END_STEP
TRANSITION FROM Check_Farbkamera TO CheckPartCam := Kamera_betriebsbereit;
END_TRANSITION
TRANSITION FROM Check_Farbkamera TO Kamera_nicht_bb := TRUE;
END_TRANSITION
STEP CheckPartCam:
END_STEP
TRANSITION FROM CheckPartCam TO Check_Abholpos_frei := NotPartCam;
END_TRANSITION
TRANSITION FROM CheckPartCam TO Robot01_Pos41 := PartCam;
END_TRANSITION
STEP Check_Abholpos_frei:
END_STEP
TRANSITION FROM Check_Abholpos_frei TO (CloseStopper, OpenSeperator) := Abholpos leer;
END_TRANSITION
TRANSITION FROM Check_Abholpos_frei TO CheckState := TRUE;
END_TRANSITION
STEP CloseStopper:
	CloseStopper_action(N);
END_STEP
STEP OpenSeperator:
	OpenSeperator_action(N);
END_STEP
TRANSITION FROM (CloseStopper, OpenSeperator) TO Wait_for_Part := State Ok;
END_TRANSITION
STEP Kamera_nicht_bb:
	Kamera_nicht_bb_entry(P1);
	Kamera_nicht_bb_action(N);
	Kamera_nicht_bb_exit(P0);
END_STEP
TRANSITION FROM Kamera_nicht_bb TO Check_Farbkamera := MsgOk;
END_TRANSITION
STEP Wait_for_Part:
	Wait_for_Part_entry(P1);
	Wait_for_Part_action(N);
	Wait_for_Part_exit(P0);
END_STEP
TRANSITION FROM Wait_for_Part TO Close_Seperator := Part Ready;
END_TRANSITION
STEP Close_Seperator:
	Close_Seperator_action(N);
END_STEP
TRANSITION FROM Close_Seperator TO Open_Stopper := StateOk;
END_TRANSITION
STEP Open_Stopper: (* min time t#500ms; t#500ms *)
	Open_Stopper_action(N);
END_STEP
TRANSITION FROM Open_Stopper TO Wait_for_Part_ := State Ok;
END_TRANSITION
STEP Wait_for_Part_:
	Wait_for_Part__entry(P1);
	Wait_for_Part__action(N);
	Wait_for_Part__exit(P0);
END_STEP
TRANSITION FROM Wait_for_Part_ TO (Close_Stopper  , Open_Seperator  ) := Part Ready;
END_TRANSITION
STEP Close_Stopper  :
	Close_Stopper  _action(N);
END_STEP
STEP Open_Seperator  :
	Open_Seperator  _action(N);
END_STEP
TRANSITION FROM (Close_Stopper  , Open_Seperator  ) TO WaitAbholPos := State Ok;
END_TRANSITION
STEP WaitAbholPos:
END_STEP
TRANSITION FROM WaitAbholPos TO GripperEmpty := AbholPos;
END_TRANSITION
STEP GripperEmpty:
END_STEP
TRANSITION FROM GripperEmpty TO CheckState := GripperEmpty;
END_TRANSITION
STEP CheckState:
END_STEP
TRANSITION FROM CheckState TO Robot01_Pos31 := #StateOK;
END_TRANSITION
STEP Robot01_Pos31: (* Pick Part / from Belt *)
	Robot01_Pos31_action(N);
	Robot01_Pos31_exit(P0);
END_STEP
TRANSITION FROM Robot01_Pos31 TO CheckCamActive := #StateOK;
END_TRANSITION
STEP CheckCamActive:
END_STEP
TRANSITION FROM CheckCamActive TO (paralellVereinzel, RobiPos) := CamActive;
END_TRANSITION
TRANSITION FROM CheckCamActive TO Result2 := TRUE;
END_TRANSITION
STEP paralellVereinzel:
END_STEP
TRANSITION FROM paralellVereinzel TO (CloseStopper_, OpenSeperator_) := Abholpos leer;
END_TRANSITION
STEP CloseStopper_:
	CloseStopper__action(N);
END_STEP
STEP OpenSeperator_:
	OpenSeperator__action(N);
END_STEP
TRANSITION FROM (CloseStopper_, OpenSeperator_) TO WaitForPart := State Ok;
END_TRANSITION
STEP WaitForPart:
	WaitForPart_entry(P1);
	WaitForPart_action(N);
	WaitForPart_exit(P0);
END_STEP
TRANSITION FROM WaitForPart TO Close_Seperator_ := Part Ready;
END_TRANSITION
TRANSITION FROM WaitForPart TO end_paralellVereinzeln := PartNotReady;
END_TRANSITION
STEP Close_Seperator_:
	Close_Seperator__action(N);
END_STEP
TRANSITION FROM Close_Seperator_ TO Open_Stopper_ := StateOk;
END_TRANSITION
STEP Open_Stopper_: (* min time t#500ms; t#500ms *)
	Open_Stopper__action(N);
END_STEP
TRANSITION FROM Open_Stopper_ TO Wait_forPart := State Ok;
END_TRANSITION
STEP Wait_forPart:
	Wait_forPart_entry(P1);
	Wait_forPart_action(N);
	Wait_forPart_exit(P0);
END_STEP
TRANSITION FROM Wait_forPart TO (Close_Stopper_  , Open_Seperator__ ) := Part Ready;
END_TRANSITION
STEP Close_Stopper_  :
	Close_Stopper_  _action(N);
END_STEP
STEP Open_Seperator__ :
	Open_Seperator__ _action(N);
END_STEP
TRANSITION FROM (Close_Stopper_  , Open_Seperator__ ) TO WaitAbholPos_ := State Ok;
END_TRANSITION
STEP WaitAbholPos_:
END_STEP
TRANSITION FROM WaitAbholPos_ TO end_paralellVereinzeln := AbholPos;
END_TRANSITION
STEP end_paralellVereinzeln:
END_STEP
STEP RobiPos:
END_STEP
TRANSITION FROM RobiPos TO Robot01_Pos41 := TRUE;
END_TRANSITION
TRANSITION FROM RobiPos TO Robot01_Pos45 := TRUE;
END_TRANSITION
STEP Robot01_Pos41: (* POS_CAM_POS1 *)
	Robot01_Pos41_entry(P1);
	Robot01_Pos41_action(N);
END_STEP
TRANSITION FROM Robot01_Pos41 TO JumpRepeat := #StateOK;
END_TRANSITION
STEP Robot01_Pos45: (* POS_CAM_POS2 *)
	Robot01_Pos45_entry(P1);
	Robot01_Pos45_action(N);
END_STEP
TRANSITION FROM Robot01_Pos45 TO JumpRepeat := #StateOK;
END_TRANSITION
STEP JumpRepeat:
END_STEP
TRANSITION FROM JumpRepeat TO (Cam1Active, Cam2Active) := TRUE;
END_TRANSITION
STEP Cam1Active:
END_STEP
TRANSITION FROM Cam1Active TO Start_Cam1 := Cam1Active;
END_TRANSITION
TRANSITION FROM Cam1Active TO ResultCam1 := TRUE;
END_TRANSITION
STEP Start_Cam1:
	Start_Cam1_action(N);
END_STEP
TRANSITION FROM Start_Cam1 TO WaitDone1 := Busy;
END_TRANSITION
STEP WaitDone1:
	WaitDone1_entry(P1);
END_STEP
TRANSITION FROM WaitDone1 TO ResultCam1_ := Done;
END_TRANSITION
STEP ResultCam1_:
	ResultCam1__entry(P1);
END_STEP
TRANSITION FROM ResultCam1_ TO EndCam1 := TRUE;
END_TRANSITION
STEP ResultCam1:
	ResultCam1_entry(P1);
END_STEP
TRANSITION FROM ResultCam1 TO EndCam1 := TRUE;
END_TRANSITION
STEP EndCam1:
END_STEP
STEP Cam2Active:
END_STEP
TRANSITION FROM Cam2Active TO Start_Cam2 := Cam2Active;
END_TRANSITION
TRANSITION FROM Cam2Active TO ResultCam2 := TRUE;
END_TRANSITION
STEP Start_Cam2:
	Start_Cam2_action(N);
END_STEP
TRANSITION FROM Start_Cam2 TO WaitDone2 := Busy;
END_TRANSITION
STEP WaitDone2:
	WaitDone2_entry(P1);
END_STEP
TRANSITION FROM WaitDone2 TO ResultCam2_ := Done;
END_TRANSITION
STEP ResultCam2_:
	ResultCam2__entry(P1);
END_STEP
TRANSITION FROM ResultCam2_ TO EndCam2 := TRUE;
END_TRANSITION
STEP ResultCam2:
	ResultCam2_entry(P1);
END_STEP
TRANSITION FROM ResultCam2 TO EndCam2 := TRUE;
END_TRANSITION
STEP EndCam2:
END_STEP
TRANSITION FROM (EndCam1, EndCam2) TO CheckPos := io;
END_TRANSITION
TRANSITION FROM (EndCam1, EndCam2) TO Result_Counter := nio;
END_TRANSITION
TRANSITION FROM (EndCam1, EndCam2) TO JumpRepeat := CheckCam1_2;
END_TRANSITION
TRANSITION FROM (EndCam1, EndCam2) TO RepeatCounter1 := CheckCam1;
END_TRANSITION
TRANSITION FROM (EndCam1, EndCam2) TO RepeatCounter2 := CheckCam2;
END_TRANSITION
STEP RepeatCounter1:
	RepeatCounter1_entry(P1);
END_STEP
TRANSITION FROM RepeatCounter1 TO Start_Cam1 := TRUE;
END_TRANSITION
STEP RepeatCounter2:
	RepeatCounter2_entry(P1);
END_STEP
TRANSITION FROM RepeatCounter2 TO Start_Cam2 := TRUE;
END_TRANSITION
STEP CheckPos:
END_STEP
TRANSITION FROM CheckPos TO checkResult := Pos = 3;
END_TRANSITION
TRANSITION FROM CheckPos TO Robot01_Pos45 := Pos = 1;
END_TRANSITION
STEP checkResult:
END_STEP
TRANSITION FROM (end_paralellVereinzeln, checkResult) TO Result_Counter := TRUE;
END_TRANSITION
STEP Result2:
	Result2_entry(P1);
END_STEP
TRANSITION FROM Result2 TO Result_Counter := TRUE;
END_TRANSITION
STEP Result_Counter:
	Result_Counter_entry(P1);
END_STEP
TRANSITION FROM Result_Counter TO SeqEnd := CounterOK;
END_TRANSITION
TRANSITION FROM Result_Counter TO Msg_Cam := Nok_Cont;
END_TRANSITION
TRANSITION FROM Result_Counter TO Msg_Cam_Percent := Nok_Percent;
END_TRANSITION
STEP Msg_Cam:
	Msg_Cam_entry(P1);
	Msg_Cam_action(N);
	Msg_Cam_exit(P0);
END_STEP
TRANSITION FROM Msg_Cam TO CounterReset := MsgOK;
END_TRANSITION
STEP CounterReset:
	CounterReset_entry(P1);
END_STEP
TRANSITION FROM CounterReset TO SeqEnd := TRUE;
END_TRANSITION
STEP Msg_Cam_Percent:
	Msg_Cam_Percent_entry(P1);
	Msg_Cam_Percent_action(N);
	Msg_Cam_Percent_exit(P0);
END_STEP
TRANSITION FROM Msg_Cam_Percent TO CounterResetP := MsgOK;
END_TRANSITION
STEP CounterResetP:
	CounterResetP_entry(P1);
END_STEP
TRANSITION FROM CounterResetP TO SeqEnd := TRUE;
END_TRANSITION
STEP SeqEnd: (* -> WAIT *)
	SeqEnd_action(N);
END_STEP
TRANSITION FROM SeqEnd TO WaitForStart := TRUE;
END_TRANSITION

ACTION Init_action:
Start:=FALSE;
State:=STATE_WAIT;
MsgOK:=FALSE;
MsgCancel:=FALSE;
SFCRun:=FALSE;
NokCounter:=0;
i:=1;
Pos:=1;
FOR i:=1 TO NO_OF_RESULT BY 1 DO
	ResultCam[i]:=RESULT_NON;
END_FOR
END_ACTION

ACTION WaitForStart_action:
IF 	Start   THEN
	State:=STATE_RUN;
	SFCTimeStart:=TIME();
	Start:=FALSE;
	FOR i:=1 TO NO_OF_RESULT BY 1 DO
		ResultCam[i]:=RESULT_NON;
	END_FOR
	i:=1;
	Pos:=1;
ELSE
	State:=STATE_WAIT;
	MsgOK:=FALSE;
	MsgCancel:=FALSE;
	SFCRun:=FALSE;
END_IF
END_ACTION

ACTION CloseStopper_action:
ST03_557_Y70_2.MoveInit:=TRUE;		(* Züführung Stopper AST/GST *)
END_ACTION

ACTION OpenSeperator_action:
ST03_557_Y70_1.MoveInit:=TRUE;		(* Zuführung Vereinzler AST/GST *)
END_ACTION

ACTION Kamera_nicht_bb_entry:
MessageHandler.ClearMessageLines(sVisu:=Visu.Message);
END_ACTION

ACTION Kamera_nicht_bb_action:
MessageHandler.Msg.ID:='PM152';
MessageHandler.Msg.Name:='Check Camera';
MessageHandler.Msg.Text:='Sesopart Kamera ist nicht betriebsbereit';
MessageHandler.Msg.Color:=Color.red;
MessageHandler.Msg.Station:=1;


MessageHandler(
	Prio:=2, 							(*1=highest, .. , 4=lowest*)
	Btn1Addr:=ADR(MsgOk),			(*Address of Button1 , if Zero then Button is unvisible*)
	Btn2Addr:=,						(*Address of Button2 , if Zero then Button is unvisible*)
	sVisu:=Visu.Message);
END_ACTION

ACTION Kamera_nicht_bb_exit:
MsgOk:=FALSE;
MsgCancel:=FALSE;
ST02_DT_95_A1.b_quitt:=TRUE;
END_ACTION

ACTION Wait_for_Part_entry:
ProcessMessage01:='';
Delay.IN:=FALSE;
Delay();
END_ACTION

ACTION Wait_for_Part_action:
ProcessMessage01:='1IM9';(*warte auf Teil in Stopper*)
Delay.IN:=ST03_556_B69_6.BitInToCheck; 		(*  ISK an Stopper.*)
Delay.PT:=T#500ms;
Delay();
END_ACTION

ACTION Wait_for_Part_exit:
ProcessMessage01:='';
END_ACTION

ACTION Close_Seperator_action:
ST03_557_Y70_1.MoveWork:=TRUE;		(*Zuführung Vereinzler AST/GST *)
END_ACTION

ACTION Open_Stopper_action:
ST03_557_Y70_2.MoveWork:=TRUE;		(* Züführung Stopper AST/GST *)
END_ACTION

ACTION Wait_for_Part__entry:
ProcessMessage01:='';
Delay(IN:=FALSE);
END_ACTION

ACTION Wait_for_Part__action:
ProcessMessage01:='1IM10';(*warte auf Teil in Abholposition*)
Delay(	IN:=	ST03_Init_AbholPos.RoboPos31,
		PT:=T#500ms);
END_ACTION

ACTION Wait_for_Part__exit:
ProcessMessage01:='';
Delay(IN:=FALSE);
END_ACTION

ACTION Close_Stopper  _action:
ST03_557_Y70_2.MoveInit:=TRUE;		(* Züführung Stopper AST/GST *)
END_ACTION

ACTION Open_Seperator  _action:
ST03_557_Y70_1.MoveInit:=TRUE;		(* Zuführung Vereinzler AST/GST *)
END_ACTION

ACTION Robot01_Pos31_action:
Robot01.PosNo:=POS_WT_POS1;
Robot01.PosOffset:=gRobotOffset;
Robot01.Override:=MP.ST00.Override;
Robot01.SetToolOn:=FALSE;
Robot01.SetToolOff:=TRUE;
Robot01.ExecuteMove:=TRUE;
END_ACTION

ACTION Robot01_Pos31_exit:
gRob01GripState:=PART_CAM;

FOR i:=1 TO NO_OF_RESULT BY 1 DO
	ResultCam[i]:=0;
END_FOR
END_ACTION

ACTION CloseStopper__action:
ST03_557_Y70_2.MoveInit:=TRUE;		(* Züführung Stopper AST/GST *)
END_ACTION

ACTION OpenSeperator__action:
ST03_557_Y70_1.MoveInit:=TRUE;		(* Zuführung Vereinzler AST/GST *)
END_ACTION

ACTION WaitForPart_entry:
ProcessMessage01:='';
Delay();
END_ACTION

ACTION WaitForPart_action:
ProcessMessage01:='1IM9';(*warte auf Teil in Stopper*)
Delay();
END_ACTION

ACTION WaitForPart_exit:
ProcessMessage01:='';
END_ACTION

ACTION Close_Seperator__action:
ST03_557_Y70_1.MoveWork:=TRUE;		(*Zuführung Vereinzler AST/GST *)
END_ACTION

ACTION Open_Stopper__action:
ST03_557_Y70_2.MoveWork:=TRUE;		(* Züführung Stopper AST/GST *)
END_ACTION

ACTION Wait_forPart_entry:
ProcessMessage01:='';
Delay(IN:=FALSE);
END_ACTION

ACTION Wait_forPart_action:
ProcessMessage01:='1IM10';(*warte auf Teil in Abholposition*)
Delay(	IN:=	ST03_Init_AbholPos.RoboPos31,
		PT:=T#500ms);
END_ACTION

ACTION Wait_forPart_exit:
ProcessMessage01:='';
Delay(IN:=FALSE);
END_ACTION

ACTION Close_Stopper_  _action:
ST03_557_Y70_2.MoveInit:=TRUE;		(* Züführung Stopper AST/GST *)
END_ACTION

ACTION Open_Seperator__ _action:
ST03_557_Y70_1.MoveInit:=TRUE;		(* Zuführung Vereinzler AST/GST *)
END_ACTION

ACTION Robot01_Pos41_entry:
RepeatCounter:=1;
END_ACTION

ACTION Robot01_Pos41_action:
Robot01.PosNo:=POS_CAM_POS1;
Robot01.PosOffset:=gRobotOffset;
Robot01.Override:=MP.ST00.Override;
Robot01.SetToolOn:=FALSE;
Robot01.SetToolOff:=TRUE;
Robot01.ExecuteMove:=TRUE;
Pos:=1;
END_ACTION

ACTION Robot01_Pos45_entry:
RepeatCounter:=0;
END_ACTION

ACTION Robot01_Pos45_action:
Robot01.PosNo:=POS_CAM_POS2;
Robot01.PosOffset:=gRobotOffset;
Robot01.Override:=MP.ST00.Override;
Robot01.SetToolOn:=FALSE;
Robot01.SetToolOff:=TRUE;
Robot01.ExecuteMove:=TRUE;
Pos:=3;
END_ACTION

ACTION Start_Cam1_action:
IF 	Pos =1 THEN
	ST03_8_100_A1.JobNo := TD.Sensopart_CamProgNo ;
ELSIF
	Pos = 3 THEN
	ST03_8_100_A1.JobNo := TD.Sensopart_CamProgNo + 1 ;
END_IF
ST03_8_100_A1.st_ctrl_in.b_start := TRUE;
END_ACTION

ACTION WaitDone1_entry:
ST03_8_100_A1.st_ctrl_in.b_start := FALSE;
RepeatCounter:=RepeatCounter+1;
END_ACTION

ACTION ResultCam1__entry:
IF 	(ST03_8_100_A1.b_Kam_Pruef_IO AND	 (*Kamera Farberkennung*)
	NOT ST03_8_100_A1.b_Kam_Pruef_NIO) OR
	CamAlwaysOK[1] THEN
	ResultCam[Pos]:=RESULT_OK;
ELSE
	ResultCam[Pos]:=RESULT_NOK;
END_IF
END_ACTION

ACTION ResultCam1_entry:
ResultCam[Pos]:=RESULT_OK;
END_ACTION

ACTION Start_Cam2_action:
IF 	Pos =1 THEN
	ST03_8_103_A1.JobNo := TD.Sensopart2_CamProgNo ;
ELSIF
	Pos = 3 THEN
	ST03_8_103_A1.JobNo := TD.Sensopart2_CamProgNo + 1 ;
END_IF
ST03_8_103_A1.st_ctrl_in.b_start := TRUE;
END_ACTION

ACTION WaitDone2_entry:
ST03_8_103_A1.st_ctrl_in.b_start := FALSE;
END_ACTION

ACTION ResultCam2__entry:
IF 	(ST03_8_103_A1.b_Kam_Pruef_IO AND	 (*Kamera Flügel*)
	NOT ST03_8_103_A1.b_Kam_Pruef_NIO) OR
	CamAlwaysOK[2] THEN
	ResultCam[Pos+1]:=RESULT_OK;
ELSE
	ResultCam[Pos+1]:=RESULT_NOK;
END_IF
END_ACTION

ACTION ResultCam2_entry:
ResultCam[Pos+1]:=RESULT_OK;
END_ACTION

ACTION RepeatCounter1_entry:
RepeatCounter:=RepeatCounter+1;
END_ACTION

ACTION RepeatCounter2_entry:
RepeatCounter:=RepeatCounter+1;
END_ACTION

ACTION Result2_entry:
FOR i:=1 TO NO_OF_RESULT BY 1 DO
	ResultCam[i]:=RESULT_OK;
END_FOR
END_ACTION

ACTION Result_Counter_entry:
FOR i:=100 TO 2 BY-1 DO
   	NokPercent[i] := NokPercent[i-1];
END_FOR

ResultOk:=TRUE;
FOR i:=1 TO NO_OF_RESULT BY 1 DO
	IF	ResultOk AND ResultCam[i] = RESULT_NOK 	THEN
		ResultOk:=FALSE;
	END_IF
END_FOR


IF 	ResultOk  THEN
	NokCounter:=0;
	NokPercent[1] := FALSE;
	gRob01GripState:=PART_OK;
ELSE
	NokCounter:=NokCounter+1;
	NokPercent[1] := TRUE;
	gRob01GripState:=PART_NOK;
END_IF
END_ACTION

ACTION Msg_Cam_entry:
MessageHandler.ClearMessageLines(sVisu:=Visu.Message);
END_ACTION

ACTION Msg_Cam_action:
MessageHandler.Msg.ID:='PM112';
MessageHandler.Msg.Name:='Sensopart Kam.-Erg. Prüfung  n.i.o:';
MessageHandler.Msg.Text:='Sensopart Kam.-Erg. Prüfung  n.i.o: Fehler in Folge';
MessageHandler.Msg.Color:=Color.red;
MessageHandler.Msg.Station:=3;
MessageHandler.MsgButton1Text:='continue';

MessageHandler(
	Prio:=2, 								(*1=highest, .. , 4=lowest*)
	Btn1Addr:=ADR(MsgOk),				(*Address of Button1 , if Zero then Button is unvisible*)
	Btn2Addr:=0(*ADR(MsgCancel)*),			(*Address of Button2 , if Zero then Button is unvisible*)
	sVisu:=Visu.Message);
END_ACTION

ACTION Msg_Cam_exit:
MsgOk:=FALSE;
MsgCancel:=FALSE;
END_ACTION

ACTION CounterReset_entry:
NokCounter:=0;
END_ACTION

ACTION Msg_Cam_Percent_entry:
MessageHandler.ClearMessageLines(sVisu:=Visu.Message);
END_ACTION

ACTION Msg_Cam_Percent_action:
MessageHandler.Msg.ID:='PM113';
MessageHandler.Msg.Name:='Sensopart Kam.-Erg. Prüfung  n.i.o:';
MessageHandler.Msg.Text:='Sensopart Kam.-Erg. Prüfung  n.i.o:% Fehler';
MessageHandler.Msg.Color:=Color.red;
MessageHandler.Msg.Station:=3;
MessageHandler.MsgButton1Text:='continue';

MessageHandler(
	Prio:=2, 								(*1=highest, .. , 4=lowest*)
	Btn1Addr:=ADR(MsgOk),				(*Address of Button1 , if Zero then Button is unvisible*)
	Btn2Addr:=0(*ADR(MsgCancel)*),			(*Address of Button2 , if Zero then Button is unvisible*)
	sVisu:=Visu.Message);
END_ACTION

ACTION Msg_Cam_Percent_exit:
MsgOk:=FALSE;
MsgCancel:=FALSE;
END_ACTION

ACTION CounterResetP_entry:
NokCounter:=0;
(*Percent Register löschen*)
FOR i:=1 TO 100 BY 1 DO
  NokPercent[i]:= FALSE;
END_FOR
END_ACTION

ACTION SeqEnd_action:
SFCTime:=TIME_TO_DINT(TIME()-SFCTimeStart);
State:=STATE_WAIT;
END_ACTION

TRANSITION Kamera_betriebsbereit:
(*Kamera Farberkennung*)
(
NOT ST03_8_100_A1.sm_kamera_nicht_bb OR
NOT ST03_8_100_A1.Activated	) AND
(
NOT ST03_8_103_A1.sm_kamera_nicht_bb OR
NOT ST03_8_103_A1.Activated	)
END_TRANSITION

TRANSITION NotPartCam:
gRob01GripState<>PART_CAM
END_TRANSITION

TRANSITION Abholpos leer:
NOT ST03_Init_AbholPos.RoboPos31
END_TRANSITION

TRANSITION PartCam:
TRUE
END_TRANSITION

TRANSITION State Ok:
ST03_557_Y70_2.State=STATE_OK AND	(*Züführung Stopper AST/GST *)
ST03_557_Y70_1.State=STATE_OK			(* Zuführung Vereinzler AST/GST *)
END_TRANSITION

TRANSITION Part Ready:
Delay.Q AND
NOT ST03_Init_AbholPos.RoboPos31 AND
ST03_556_B69_6.BitInToCheck	AND			(*ISK anwesend am Stoper*)
Robot01.ActualArea <> 4
END_TRANSITION

TRANSITION StateOk:
ST03_557_Y70_1.State=STATE_OK AND	(* Zuführung Vereinzler AST/GST *)
Robot01.ActualArea <> 4
END_TRANSITION

TRANSITION State Ok:
ST03_557_Y70_2.State=STATE_OK 	(* Züführung Stopper AST/GST *)
END_TRANSITION

TRANSITION Part Ready:
Delay.Q AND
Robot01.ActualArea <> 4
END_TRANSITION

TRANSITION State Ok:
ST03_557_Y70_2.State=STATE_OK AND	(*Züführung Stopper AST/GST *)
ST03_557_Y70_1.State=STATE_OK			(* Zuführung Vereinzler AST/GST *)
END_TRANSITION

TRANSITION AbholPos:
ST03_Init_AbholPos.RoboPos31 	(*ISK  auf Übergabeposition *)
END_TRANSITION

TRANSITION GripperEmpty:
gRob01GripState=PART_NO AND
Robot01.RemInToolWorkSensor
END_TRANSITION

TRANSITION #StateOK:
Robot01.State=STATE_WAIT AND
gRob01GripState=PART_NO
END_TRANSITION

TRANSITION #StateOK:
Robot01.State=STATE_OK AND
gTipImp
END_TRANSITION

TRANSITION CamActive:
ST03_8_100_A1.Activated OR
ST03_8_103_A1.Activated
END_TRANSITION

TRANSITION Abholpos leer:
NOT ST03_Init_AbholPos.RoboPos31 AND
Robot01.ActualArea <> 4
END_TRANSITION

TRANSITION State Ok:
ST03_557_Y70_2.State=STATE_OK AND	(*Züführung Stopper AST/GST *)
ST03_557_Y70_1.State=STATE_OK			(* Zuführung Vereinzler AST/GST *)
END_TRANSITION

TRANSITION Part Ready:
NOT ST03_Init_AbholPos.RoboPos31 AND
ST03_556_B69_6.BitInToCheck	AND			(*ISK anwesend am Stoper*)
Robot01.ActualArea <> 4
END_TRANSITION

TRANSITION StateOk:
ST03_557_Y70_1.State=STATE_OK AND	(* Zuführung Vereinzler AST/GST *)
Robot01.ActualArea <> 4
END_TRANSITION

TRANSITION State Ok:
ST03_557_Y70_2.State=STATE_OK 	(* Züführung Stopper AST/GST *)
END_TRANSITION

TRANSITION Part Ready:
Delay.Q AND
Robot01.ActualArea <> 4
END_TRANSITION

TRANSITION State Ok:
ST03_557_Y70_2.State=STATE_OK AND	(*Züführung Stopper AST/GST *)
ST03_557_Y70_1.State=STATE_OK			(* Zuführung Vereinzler AST/GST *)
END_TRANSITION

TRANSITION AbholPos:
ST03_Init_AbholPos.RoboPos31 	(*ISK  auf Übergabeposition *)
END_TRANSITION

TRANSITION PartNotReady:
NOT ST03_556_B69_6.BitInToCheck 		(*  ISK an Stopper.*)
END_TRANSITION

TRANSITION #StateOK:
Robot01.State=STATE_OK AND
gTipImp
END_TRANSITION

TRANSITION #StateOK:
Robot01.State=STATE_OK AND
gTipImp
END_TRANSITION

TRANSITION Cam1Active:
ST03_8_100_A1.Activated
END_TRANSITION

TRANSITION Busy:
ST03_8_100_A1.st_ctrl_out.b_busy (*Kamera Farberkennung Ehternet*)
END_TRANSITION

TRANSITION Done:
ST03_8_100_A1.st_ctrl_out.b_fertig
END_TRANSITION

TRANSITION Cam2Active:
ST03_8_103_A1.Activated
END_TRANSITION

TRANSITION Busy:
ST03_8_103_A1.st_ctrl_out.b_busy (*Kamera Farberkennung Ehternet*)
END_TRANSITION

TRANSITION Done:
ST03_8_103_A1.st_ctrl_out.b_fertig
END_TRANSITION

TRANSITION io:
ResultCam[Pos]=RESULT_OK AND
ResultCam[Pos+1]=RESULT_OK
END_TRANSITION

TRANSITION nio:
RepeatCounter>=2
END_TRANSITION

TRANSITION CheckCam1_2:
ResultCam[Pos]=RESULT_NOK AND
ResultCam[Pos+1]=RESULT_NOK
END_TRANSITION

TRANSITION CheckCam1:
ResultCam[Pos]=RESULT_NOK
END_TRANSITION

TRANSITION CheckCam2:
ResultCam[Pos+1]=RESULT_NOK
END_TRANSITION

TRANSITION CounterOK:
NokCounter<MP.ST03.CamNoOfErrors AND
NokCounterPercent < MP.ST02.CamNoOfErrorsPercent
END_TRANSITION

TRANSITION Nok_Cont:
NokCounter >= MP.ST03.CamNoOfErrors
END_TRANSITION

TRANSITION Nok_Percent:
NokCounterPercent >= MP.ST03.CamNoOfErrorsPercent
END_TRANSITION
END_PROGRAM

(* POU Stations/ST_03_Ruestsaetze/ST_03_SFCs/Zufuehrungen/ST03_268_RP_Zufuehrung, SFC *)
 PROGRAM ST03_268_RP_Zufuehrung
VAR_OUTPUT
	SFCCurrentPOU			: STRING:='ST03_268_RP_Zufuehrung';
	SFCCurrentStep			: STRING:='';
	FB_CurrentStepHistorie	:FB_CurrentStepHistorie;
	SFCTime					: DINT;
	State   				: StateObject	:= STATE_WAIT;
	Result  				: StateResult;
END_VAR
VAR_INPUT
	Start					:BOOL;
END_VAR
VAR
	MsgOK				: BOOL;
	MsgCancel			: BOOL;
	SFCRun			: BOOL;
	SFCTimeStart		: TIME;
	Delay				: TON;
	Delay2				: TON;
	(* Userdefinded area *)

END_VAR
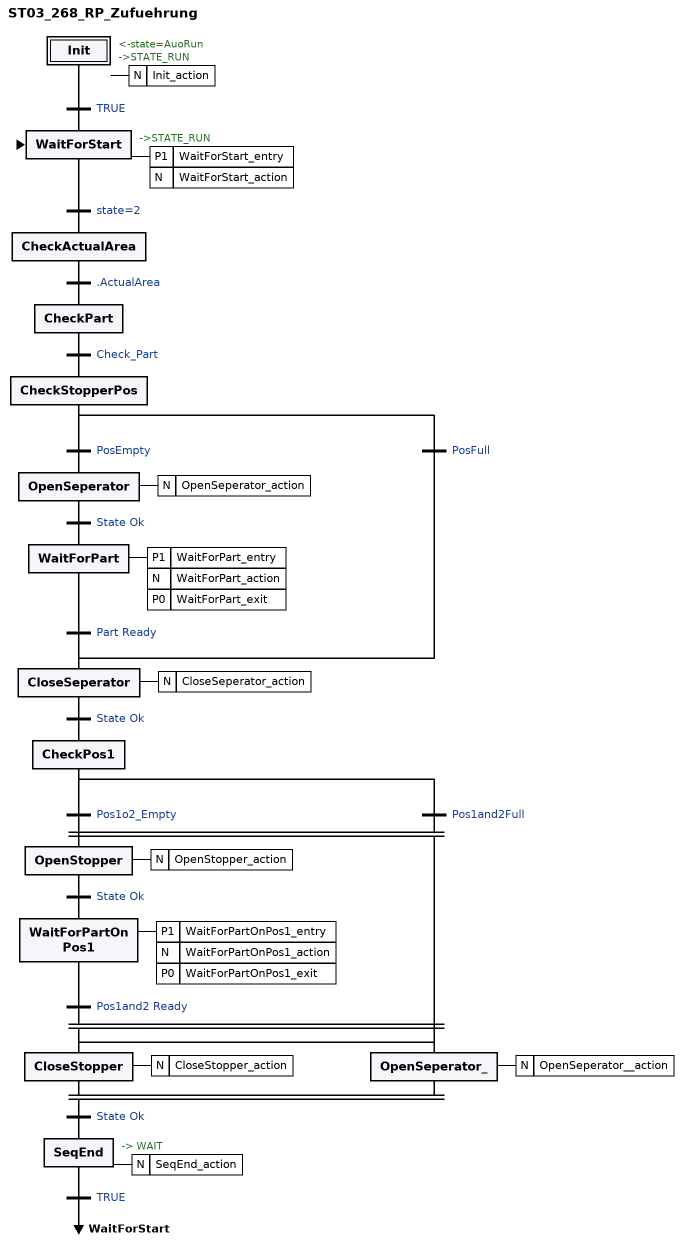
INITIAL_STEP Init: (* <-state=AuoRun / ->STATE_RUN *)
	Init_action(N);
END_STEP
TRANSITION FROM Init TO WaitForStart := TRUE;
END_TRANSITION
STEP WaitForStart: (* ->STATE_RUN *)
	WaitForStart_entry(P1);
	WaitForStart_action(N);
END_STEP
TRANSITION FROM WaitForStart TO CheckActualArea  := state=2;
END_TRANSITION
STEP CheckActualArea :
END_STEP
TRANSITION FROM CheckActualArea  TO CheckPart := .ActualArea;
END_TRANSITION
STEP CheckPart:
END_STEP
TRANSITION FROM CheckPart TO CheckStopperPos := Check_Part;
END_TRANSITION
STEP CheckStopperPos:
END_STEP
TRANSITION FROM CheckStopperPos TO OpenSeperator := PosEmpty;
END_TRANSITION
TRANSITION FROM CheckStopperPos TO CloseSeperator := PosFull;
END_TRANSITION
STEP OpenSeperator:
	OpenSeperator_action(N);
END_STEP
TRANSITION FROM OpenSeperator TO WaitForPart := State Ok;
END_TRANSITION
STEP WaitForPart:
	WaitForPart_entry(P1);
	WaitForPart_action(N);
	WaitForPart_exit(P0);
END_STEP
TRANSITION FROM WaitForPart TO CloseSeperator := Part Ready;
END_TRANSITION
STEP CloseSeperator:
	CloseSeperator_action(N);
END_STEP
TRANSITION FROM CloseSeperator TO CheckPos1 := State Ok;
END_TRANSITION
STEP CheckPos1:
END_STEP
TRANSITION FROM CheckPos1 TO OpenStopper := Pos1o2_Empty;
END_TRANSITION
TRANSITION FROM CheckPos1 TO (CloseStopper, OpenSeperator_) := Pos1and2Full;
END_TRANSITION
STEP OpenStopper:
	OpenStopper_action(N);
END_STEP
TRANSITION FROM OpenStopper TO WaitForPartOnPos1 := State Ok;
END_TRANSITION
STEP WaitForPartOnPos1:
	WaitForPartOnPos1_entry(P1);
	WaitForPartOnPos1_action(N);
	WaitForPartOnPos1_exit(P0);
END_STEP
TRANSITION FROM WaitForPartOnPos1 TO (CloseStopper, OpenSeperator_) := Pos1and2 Ready;
END_TRANSITION
STEP CloseStopper:
	CloseStopper_action(N);
END_STEP
STEP OpenSeperator_:
	OpenSeperator__action(N);
END_STEP
TRANSITION FROM (CloseStopper, OpenSeperator_) TO SeqEnd := State Ok;
END_TRANSITION
STEP SeqEnd: (* -> WAIT *)
	SeqEnd_action(N);
END_STEP
TRANSITION FROM SeqEnd TO WaitForStart := TRUE;
END_TRANSITION

ACTION Init_action:
Start:=FALSE;
State:=STATE_WAIT;
MsgOK:=FALSE;
MsgCancel:=FALSE;
SFCRun:=FALSE;
Result:=RESULT_NON;
END_ACTION

ACTION WaitForStart_entry:
;
END_ACTION

ACTION WaitForStart_action:
IF 	Start   THEN
	State:=STATE_RUN;
	Result:=RESULT_NON;
	SFCTimeStart:=TIME();
	Start:=FALSE;
ELSE
	State:=STATE_WAIT;
	MsgOK:=FALSE;
	MsgCancel:=FALSE;
	SFCRun:=FALSE;
END_IF
END_ACTION

ACTION OpenSeperator_action:
ST03_564_Y71_0.MoveInit:=TRUE;		(*Zuführung 1 Vereinzler AST/GST *)
ST03_564_Y71_2.MoveInit:=TRUE;		(*Zuführung 2 Vereinzler AST/GST *)
END_ACTION

ACTION WaitForPart_entry:
ProcessMessage02:='';
Delay(IN:=FALSE);
END_ACTION

ACTION WaitForPart_action:
ProcessMessage02:='2IM6';						(*warte auf Teil Übergabeposition 1*)
END_ACTION

ACTION WaitForPart_exit:
ProcessMessage02:='';
END_ACTION

ACTION CloseSeperator_action:
ST03_564_Y71_0.MoveWork:=TRUE;		(*Zuführung 1 Vereinzler AST/GST *)
ST03_564_Y71_2.MoveWork:=TRUE;		(*Zuführung 2 Vereinzler AST/GST *)
END_ACTION

ACTION OpenStopper_action:
IF 	NOT ST03_562_B67_7.BitInToCheck THEN	(*Zuführung 1 ISK auf Übergabepos. Robi*)
	ST03_564_Y71_1.MoveWork:=TRUE;		(*Zuführung 1 Stopper AST/GST *)
END_IF
IF 	NOT ST03_563_B70_7.BitInToCheck THEN	 (*Zuführung 2 ISK auf Übergabepos. Robi*)
	ST03_564_Y71_3.MoveWork:=TRUE;		(*Zuführung 2 Stopper AST/GST *)
END_IF
END_ACTION

ACTION WaitForPartOnPos1_entry:
ProcessMessage02:='';
Delay(IN:=FALSE);
END_ACTION

ACTION WaitForPartOnPos1_action:
ProcessMessage02:='2IM6';						(*warte auf Teil Übergabeposition 1*)
END_ACTION

ACTION WaitForPartOnPos1_exit:
ProcessMessage02:='';
END_ACTION

ACTION CloseStopper_action:
ST03_564_Y71_1.MoveInit:=TRUE;		(*Zuführung 1 Stopper AST/GST *)
ST03_564_Y71_3.MoveInit:=TRUE;		(*Zuführung 2 Stopper AST/GST *)
END_ACTION

ACTION OpenSeperator__action:
IF	NOT ST03_562_B69_6.BitInToCheck	THEN 	(*  ISK 1 anwesend am Stopper*)
	ST03_564_Y71_0.MoveInit:=TRUE;			(*Zuführung 1 Vereinzler AST/GST *)
END_IF
IF	NOT ST03_563_B70_6.BitInToCheck	THEN	 (*  ISK 2 anwesend am Stopper*)
	ST03_564_Y71_2.MoveInit:=TRUE;			(*Zuführung 2 Vereinzler AST/GST *)
END_IF
END_ACTION

ACTION SeqEnd_action:
SFCTime:=TIME_TO_DINT(TIME()-SFCTimeStart);
State:=STATE_WAIT;
END_ACTION

TRANSITION .ActualArea:
Robot01.ActualArea <> 4
END_TRANSITION

TRANSITION Check_Part:
NOT ST03_513_B70_7.BitInToCheck OR	(* ISK auf Übergabeposition  1*)
NOT ST03_514_B71_2.BitInToCheck OR	(* ISK auf Übergabeposition  2*)
NOT ST03_514_B71_5.BitInToCheck OR	(* ISK auf Übergabeposition  3*)
NOT ST03_514_B71_6.BitInToCheck		(* ISK auf Übergabeposition  4*)
END_TRANSITION

TRANSITION PosEmpty:
NOT ST03_562_B69_6.BitInToCheck	OR	 	(*  ISK 1 anwesend am Stopper*)
NOT ST03_563_B70_6.BitInToCheck		 	(*  ISK 2 anwesend am Stopper*)
END_TRANSITION

TRANSITION State Ok:
ST03_564_Y71_0.State=STATE_OK AND	(*Zuführung 1 Vereinzler AST/GST *)
ST03_564_Y71_2.State=STATE_OK 		(*Zuführung 2 Vereinzler AST/GST *)
END_TRANSITION

TRANSITION Part Ready:
ST03_562_B69_6.BitInToCheck	AND	(*  ISK 1 anwesend am Stopper*)
ST03_563_B70_6.BitInToCheck		 	(*  ISK 2 anwesend am Stopper*)
END_TRANSITION

TRANSITION PosFull:
ST03_562_B69_6.BitInToCheck	AND	 	(*  ISK 1 anwesend am Stopper*)
ST03_563_B70_6.BitInToCheck			 	(*  ISK 2 anwesend am Stopper*)
END_TRANSITION

TRANSITION State Ok:
ST03_564_Y71_0.State=STATE_OK AND	(*Zuführung 1 Vereinzler AST/GST *)
ST03_564_Y71_2.State=STATE_OK 		(*Zuführung 2 Vereinzler AST/GST *)
END_TRANSITION

TRANSITION Pos1o2_Empty:
NOT ST03_562_B67_7.BitInToCheck OR	(*Zuführung 1 ISK auf Übergabepos. Robi*)
NOT ST03_563_B70_7.BitInToCheck	 	(*Zuführung 2 ISK auf Übergabepos. Robi*)
END_TRANSITION

TRANSITION State Ok:
ST03_564_Y71_1.State=STATE_OK AND 	(*Zuführung 1 Stopper AST/GST *)
ST03_564_Y71_3.State=STATE_OK 		(*Zuführung 2 Stopper AST/GST *)
END_TRANSITION

TRANSITION Pos1and2 Ready:
ST03_562_B67_7.BitInToCheck 	AND	 (*Zuführung 1 ISK auf Übergabepos. Robi*)
ST03_563_B70_7.BitInToCheck 			 (*Zuführung 2 ISK auf Übergabepos. Robi*)
END_TRANSITION

TRANSITION Pos1and2Full:
ST03_562_B67_7.BitInToCheck AND	(*Zuführung 1 ISK auf Übergabepos. Robi*)
ST03_563_B70_7.BitInToCheck	 	(*Zuführung 2 ISK auf Übergabepos. Robi*)
END_TRANSITION

TRANSITION State Ok:
ST03_564_Y71_1.State=STATE_OK 	AND	(*Zuführung 1 Stopper AST/GST *)
ST03_564_Y71_3.State=STATE_OK 		(*Zuführung 2 Stopper AST/GST *)
END_TRANSITION
END_PROGRAM

(* POU Stations/ST_03_Ruestsaetze/ST_03_SFCs/Zufuehrungen/ST03_268_RP_Wendeeinheit, SFC *)
 PROGRAM ST03_268_RP_Wendeeinheit

VAR_OUTPUT
	SFCCurrentPOU			: STRING:='ST03_268_RP_Wendeeinheit';
	SFCCurrentStep			: STRING:='';
	FB_CurrentStepHistorie	: FB_CurrentStepHistorie;
	SFCTime					: DINT;
	State   				: StateObject	:= STATE_WAIT;
	Result  				: StateResult;

END_VAR
VAR_INPUT
	Start				:BOOL;
END_VAR
VAR
	MsgOK				: BOOL;
	MsgCancel			: BOOL;
	SFCRun				: BOOL;
	SFCTimeStart		: TIME;
	Delay				: TON;
	(* Userdefinded area *)
	WenderDone			: BOOL;
	OverrideHelp			:DINT;
END_VAR
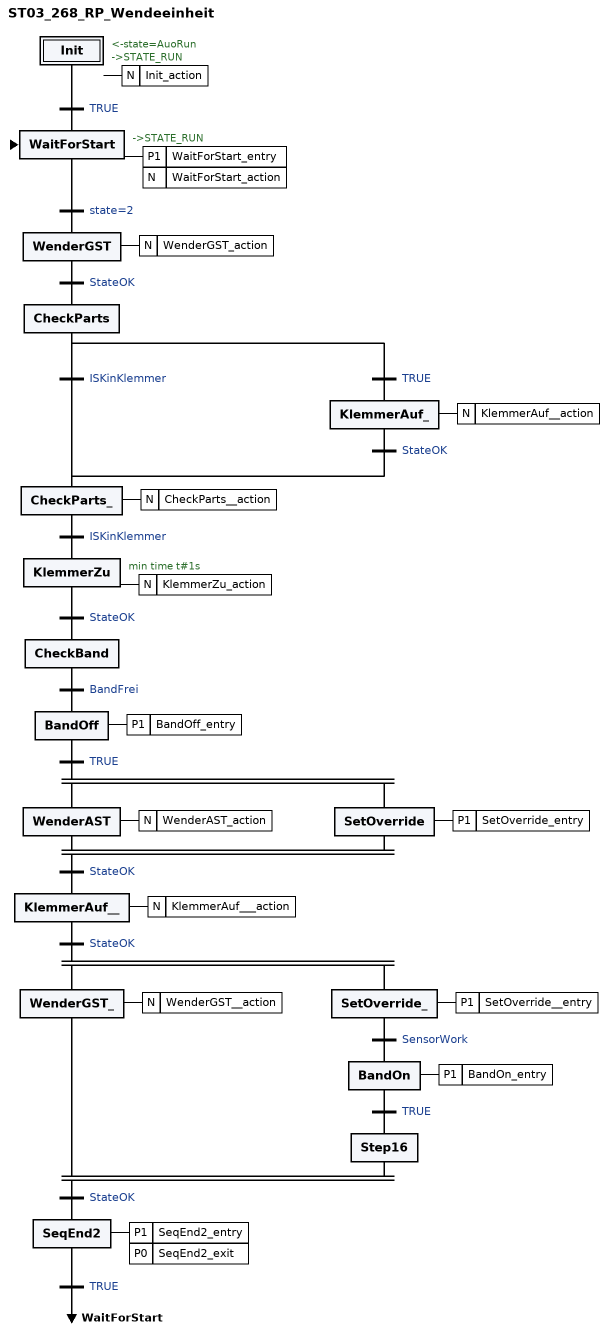
INITIAL_STEP Init: (* <-state=AuoRun / ->STATE_RUN *)
	Init_action(N);
END_STEP
TRANSITION FROM Init TO WaitForStart := TRUE;
END_TRANSITION
STEP WaitForStart: (* ->STATE_RUN *)
	WaitForStart_entry(P1);
	WaitForStart_action(N);
END_STEP
TRANSITION FROM WaitForStart TO WenderGST := state=2;
END_TRANSITION
STEP WenderGST:
	WenderGST_action(N);
END_STEP
TRANSITION FROM WenderGST TO CheckParts := StateOK;
END_TRANSITION
STEP CheckParts:
END_STEP
TRANSITION FROM CheckParts TO CheckParts_ := ISKinKlemmer;
END_TRANSITION
TRANSITION FROM CheckParts TO KlemmerAuf_ := TRUE;
END_TRANSITION
STEP KlemmerAuf_:
	KlemmerAuf__action(N);
END_STEP
TRANSITION FROM KlemmerAuf_ TO CheckParts_ := StateOK;
END_TRANSITION
STEP CheckParts_:
	CheckParts__action(N);
END_STEP
TRANSITION FROM CheckParts_ TO KlemmerZu := ISKinKlemmer;
END_TRANSITION
STEP KlemmerZu: (* min time t#1s *)
	KlemmerZu_action(N);
END_STEP
TRANSITION FROM KlemmerZu TO CheckBand := StateOK;
END_TRANSITION
STEP CheckBand:
END_STEP
TRANSITION FROM CheckBand TO BandOff := BandFrei;
END_TRANSITION
STEP BandOff:
	BandOff_entry(P1);
END_STEP
TRANSITION FROM BandOff TO (WenderAST, SetOverride) := TRUE;
END_TRANSITION
STEP WenderAST:
	WenderAST_action(N);
END_STEP
STEP SetOverride:
	SetOverride_entry(P1);
END_STEP
TRANSITION FROM (WenderAST, SetOverride) TO KlemmerAuf__ := StateOK;
END_TRANSITION
STEP KlemmerAuf__:
	KlemmerAuf___action(N);
END_STEP
TRANSITION FROM KlemmerAuf__ TO (WenderGST_, SetOverride_) := StateOK;
END_TRANSITION
STEP WenderGST_:
	WenderGST__action(N);
END_STEP
STEP SetOverride_:
	SetOverride__entry(P1);
END_STEP
TRANSITION FROM SetOverride_ TO BandOn := SensorWork;
END_TRANSITION
STEP BandOn:
	BandOn_entry(P1);
END_STEP
TRANSITION FROM BandOn TO Step16 := TRUE;
END_TRANSITION
STEP Step16:
END_STEP
TRANSITION FROM (WenderGST_, Step16) TO SeqEnd2 := StateOK;
END_TRANSITION
STEP SeqEnd2:
	SeqEnd2_entry(P1);
	SeqEnd2_exit(P0);
END_STEP
TRANSITION FROM SeqEnd2 TO WaitForStart := TRUE;
END_TRANSITION

ACTION Init_action:
Start:=FALSE;
State:=STATE_WAIT;
MsgOK:=FALSE;
MsgCancel:=FALSE;
SFCRun:=FALSE;
Result:=RESULT_NON;
IF 	OverrideHelp <> 0 THEN
	MP.ST02.Override_Band:=OverrideHelp;
END_IF

ST03_Band.bLockBand := FALSE;
END_ACTION

ACTION WaitForStart_entry:
;
END_ACTION

ACTION WaitForStart_action:
IF 	Start   THEN
	State:=STATE_RUN;
	Result:=RESULT_NON;
	SFCTimeStart:=TIME();
	Start:=FALSE;
	WenderDone:=FALSE;
ELSE
	State:=STATE_WAIT;
	MsgOK:=FALSE;
	MsgCancel:=FALSE;
	SFCRun:=FALSE;
END_IF
END_ACTION

ACTION WenderGST_action:
ST03_564_Y71_5.MoveInit:=TRUE;		(* Rinne schwenkern AST/GST *)
END_ACTION

ACTION KlemmerAuf__action:
ST03_564_Y71_4.MoveInit:=TRUE;		(* ISK Klemmer AST/GST *)
END_ACTION

ACTION CheckParts__action:
ProcessMessage01:='1IM6';						(*'warte auf Teil in Vereinzelung*)
END_ACTION

ACTION KlemmerZu_action:
ST03_564_Y71_4.MoveWork:=TRUE;		(* ISK Klemmer AST/GST *)
END_ACTION

ACTION BandOff_entry:
ST03_Band.bLockBand := TRUE;
END_ACTION

ACTION WenderAST_action:
ST03_564_Y71_5.MoveWork:=TRUE;		(* Rinne schwenkern AST/GST *)
END_ACTION

ACTION SetOverride_entry:
IF 	MP.ST02.Override_Band > 20 THEN
	OverrideHelp:=MP.ST02.Override_Band;
	MP.ST02.Override_Band:= 15;
END_IF
END_ACTION

ACTION KlemmerAuf___action:
ST03_564_Y71_4.MoveInit:=TRUE;	(* ISK Klemmer AST/GST *)
END_ACTION

ACTION WenderGST__action:
ST03_564_Y71_5.MoveInit:=TRUE;		(* Rinne schwenkern AST/GST *)
END_ACTION

ACTION SetOverride__entry:
MP.ST02.Override_Band:=OverrideHelp;
END_ACTION

ACTION BandOn_entry:
ST03_Band.bLockBand := FALSE;
END_ACTION

ACTION SeqEnd2_entry:
WenderDone:=TRUE;
END_ACTION

ACTION SeqEnd2_exit:
WenderDone:=FALSE;
END_ACTION

TRANSITION StateOK:
ST03_564_Y71_5.State = STATE_OK 	(* Rinne schwenkern AST/GST *)
END_TRANSITION

TRANSITION ISKinKlemmer:
ST03_565_B72_0.BitInToCheck AND	(* ISK 1 in Klemmer *)
ST03_565_B72_1.BitInToCheck 		(* ISK 2 in Klemmer *)
END_TRANSITION

TRANSITION StateOK:
ST03_564_Y71_4.State = STATE_OK		(*   ISK Klemmer AST/GST *)
END_TRANSITION

TRANSITION ISKinKlemmer:
ST03_565_B72_0.BitInToCheck AND 	(* ISK 1 in Klemmer *)
ST03_565_B72_1.BitInToCheck AND 	(* ISK 2 in Klemmer *)
(ST00_73_K4.BitInToCheck 	OR ST02_S1_40K01.BitInToCheck)		(*Schnittstelle Freigabe von Spritzmaschine (nur für Anlagen ohne Rundtisch)*)
END_TRANSITION

TRANSITION StateOK:
ST03_564_Y71_4.State = STATE_OK			(* ISK Klemmer AST/GST *)
END_TRANSITION

TRANSITION BandFrei:
ST03_562_B69_0.BitInToCheck  AND	(*Zuführung 1 frei zum schwenken*)
ST03_563_B70_0.BitInToCheck 	 	(*Zuführung 2 frei zum schwenken*)
END_TRANSITION

TRANSITION StateOK:
ST03_564_Y71_5.State = STATE_OK 	(* Förderband  Zuführung Vereinzelner Wender AST/GST *)
END_TRANSITION

TRANSITION StateOK:
ST03_564_Y71_4.State = STATE_OK	(* ISK Klemmer AST/GST *)
END_TRANSITION

TRANSITION SensorWork:
NOT ST03_564_Y71_5.SensorWorkIn[1].SensorSignal
END_TRANSITION

TRANSITION StateOK:
ST03_564_Y71_5.State = STATE_OK 	(* Rinne schwenkern AST/GST *)
END_TRANSITION
END_PROGRAM

(* POU Stations/ST_03_Ruestsaetze/ST_03_SFCs/Zufuehrungen/ST03_91pol_Zufuehrung, SFC *)
 PROGRAM ST03_91pol_Zufuehrung
VAR_OUTPUT
	SFCCurrentPOU		: STRING:='ST03_21pol_Zufuehrung';
	SFCCurrentStep		: STRING:='';
	FB_CurrentStepHistorie: FB_CurrentStepHistorie;
	SFCTime				: DINT;
	State   			: StateObject	:= STATE_WAIT;
	Result  			: StateResult;
END_VAR
VAR_INPUT
	Start				:BOOL;
END_VAR
VAR
	MsgOK				: BOOL;
	MsgCancel			: BOOL;
	SFCRun				: BOOL;
	SFCTimeStart		: TIME;
	Delay				: TON;
	(* Userdefinded area *)

END_VAR
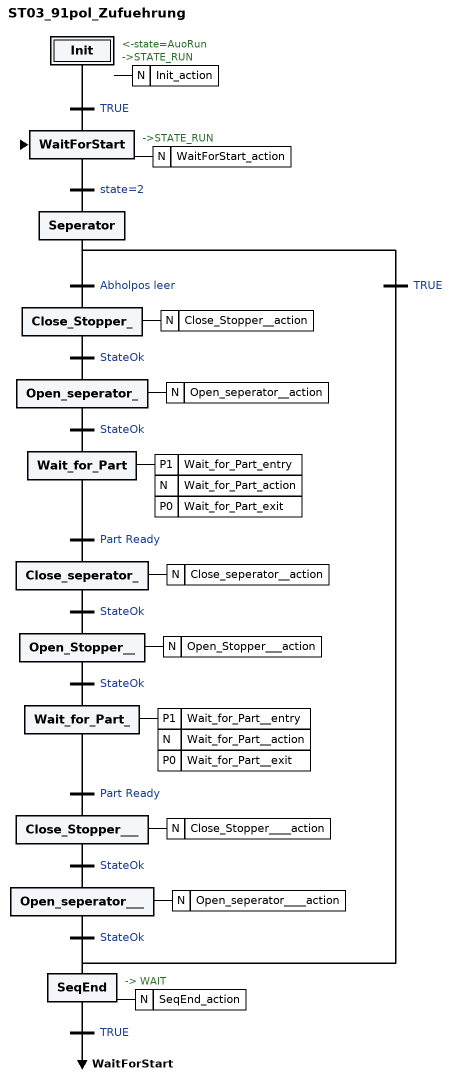
INITIAL_STEP Init: (* <-state=AuoRun / ->STATE_RUN *)
	Init_action(N);
END_STEP
TRANSITION FROM Init TO WaitForStart := TRUE;
END_TRANSITION
STEP WaitForStart: (* ->STATE_RUN *)
	WaitForStart_action(N);
END_STEP
TRANSITION FROM WaitForStart TO Seperator := state=2;
END_TRANSITION
STEP Seperator:
END_STEP
TRANSITION FROM Seperator TO Close_Stopper_ := Abholpos leer;
END_TRANSITION
TRANSITION FROM Seperator TO SeqEnd := TRUE;
END_TRANSITION
STEP Close_Stopper_:
	Close_Stopper__action(N);
END_STEP
TRANSITION FROM Close_Stopper_ TO Open_seperator_ := StateOk;
END_TRANSITION
STEP Open_seperator_:
	Open_seperator__action(N);
END_STEP
TRANSITION FROM Open_seperator_ TO Wait_for_Part := StateOk;
END_TRANSITION
STEP Wait_for_Part:
	Wait_for_Part_entry(P1);
	Wait_for_Part_action(N);
	Wait_for_Part_exit(P0);
END_STEP
TRANSITION FROM Wait_for_Part TO Close_seperator_ := Part Ready;
END_TRANSITION
STEP Close_seperator_:
	Close_seperator__action(N);
END_STEP
TRANSITION FROM Close_seperator_ TO Open_Stopper__ := StateOk;
END_TRANSITION
STEP Open_Stopper__:
	Open_Stopper___action(N);
END_STEP
TRANSITION FROM Open_Stopper__ TO Wait_for_Part_ := StateOk;
END_TRANSITION
STEP Wait_for_Part_:
	Wait_for_Part__entry(P1);
	Wait_for_Part__action(N);
	Wait_for_Part__exit(P0);
END_STEP
TRANSITION FROM Wait_for_Part_ TO Close_Stopper___ := Part Ready;
END_TRANSITION
STEP Close_Stopper___:
	Close_Stopper____action(N);
END_STEP
TRANSITION FROM Close_Stopper___ TO Open_seperator___ := StateOk;
END_TRANSITION
STEP Open_seperator___:
	Open_seperator____action(N);
END_STEP
TRANSITION FROM Open_seperator___ TO SeqEnd := StateOk;
END_TRANSITION
STEP SeqEnd: (* -> WAIT *)
	SeqEnd_action(N);
END_STEP
TRANSITION FROM SeqEnd TO WaitForStart := TRUE;
END_TRANSITION

ACTION Init_action:
Start:=FALSE;
State:=STATE_WAIT;
MsgOK:=FALSE;
MsgCancel:=FALSE;
SFCRun:=FALSE;
Result:=RESULT_NON;
END_ACTION

ACTION WaitForStart_action:
IF 	Start   THEN
	State:=STATE_RUN;
	Result:=RESULT_NON;
	SFCTimeStart:=TIME();
	Start:=FALSE;
ELSE
	State:=STATE_WAIT;
	MsgOK:=FALSE;
	MsgCancel:=FALSE;
	SFCRun:=FALSE;
END_IF
END_ACTION

ACTION Close_Stopper__action:
ST08_412_Y55_2.MoveWork:=TRUE;
END_ACTION

ACTION Open_seperator__action:
ST08_412_Y55_0.MoveInit:=TRUE;
END_ACTION

ACTION Wait_for_Part_entry:
ProcessMessage01:='';
Delay.IN:=FALSE;
Delay();
END_ACTION

ACTION Wait_for_Part_action:
ProcessMessage01:='1IM9';(*warte auf Teil in Stopper*)
Delay.IN:=ST08_412_B58_7.BitInToCheck;	(*  ISK an stopper.*)
Delay.PT:=T#50ms;
Delay();
END_ACTION

ACTION Wait_for_Part_exit:
ProcessMessage01:='';
END_ACTION

ACTION Close_seperator__action:
ST08_412_Y55_0.MoveWork:=TRUE;
END_ACTION

ACTION Open_Stopper___action:
ST08_412_Y55_2.MoveInit:=TRUE;
END_ACTION

ACTION Wait_for_Part__entry:
ProcessMessage01:='';
Delay.IN:=FALSE;
Delay();
END_ACTION

ACTION Wait_for_Part__action:
ProcessMessage01:='1IM10';(*warte auf Teil in Abholposition*)
Delay.IN:=	ST03_Init_AbholPos.RoboPos31 OR
			ST03_Init_AbholPos.RoboPos35;
Delay.PT:=T#50ms;
Delay();
END_ACTION

ACTION Wait_for_Part__exit:
ProcessMessage01:='';
END_ACTION

ACTION Close_Stopper____action:
ST08_412_Y55_2.MoveWork:=TRUE;
END_ACTION

ACTION Open_seperator____action:
ST08_412_Y55_0.MoveInit:=TRUE;
END_ACTION

ACTION SeqEnd_action:
SFCTime:=TIME_TO_DINT(TIME()-SFCTimeStart);
State:=STATE_WAIT;
END_ACTION

TRANSITION Abholpos leer:
NOT ST08_412_B59_0.BitInToCheck 		 (* Teil auf Abholpos *)
END_TRANSITION

TRANSITION StateOk:
ST08_412_Y55_2.State=STATE_OK
END_TRANSITION

TRANSITION StateOk:
ST08_412_Y55_0.State=STATE_OK
END_TRANSITION

TRANSITION Part Ready:
Delay.Q AND
Robot01.ActualArea <> 4
END_TRANSITION

TRANSITION StateOk:
ST08_412_Y55_0.State=STATE_OK
END_TRANSITION

TRANSITION StateOk:
ST08_412_Y55_2.State=STATE_OK
END_TRANSITION

TRANSITION Part Ready:
Delay.Q AND
Robot01.ActualArea <> 4
END_TRANSITION

TRANSITION StateOk:
ST08_412_Y55_2.State=STATE_OK
END_TRANSITION

TRANSITION StateOk:
ST08_412_Y55_0.State=STATE_OK
END_TRANSITION
END_PROGRAM

(* POU Stations/ST_03_Ruestsaetze/ST_03_SFCs/Zufuehrungen/ST03_33pol_Zufuehrung, SFC *)
 PROGRAM ST03_33pol_Zufuehrung
VAR_OUTPUT
	SFCCurrentPOU			: STRING:='ST03_33pol_Zufuehrung';
	SFCCurrentStep			: STRING:='';
	FB_CurrentStepHistorie:FB_CurrentStepHistorie;
	SFCTime					: DINT;
	State   				: StateObject	:= STATE_WAIT;
	Result  				: StateResult;
END_VAR
VAR_INPUT
	Start					:BOOL;
END_VAR
VAR
	MsgOK				: BOOL;
	MsgCancel			: BOOL;
	SFCRun				: BOOL;
	SFCTimeStart		: TIME;
	Delay				: TON;
	(* Userdefinded area *)

END_VAR
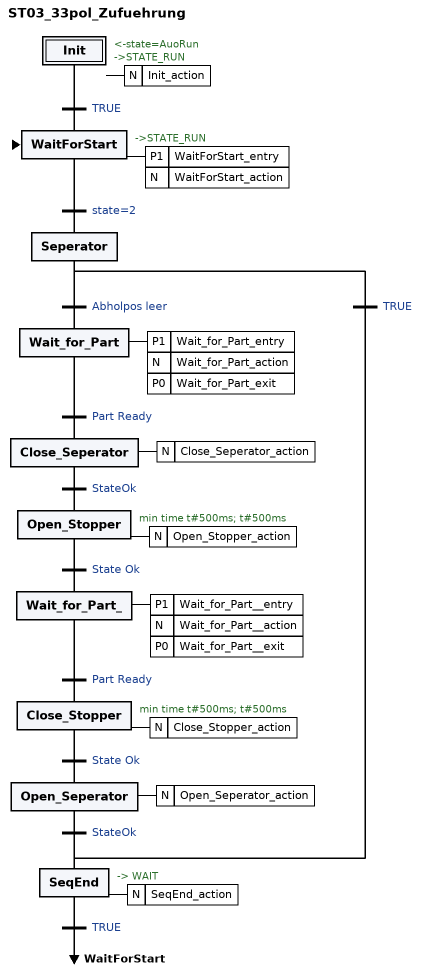
INITIAL_STEP Init: (* <-state=AuoRun / ->STATE_RUN *)
	Init_action(N);
END_STEP
TRANSITION FROM Init TO WaitForStart := TRUE;
END_TRANSITION
STEP WaitForStart: (* ->STATE_RUN *)
	WaitForStart_entry(P1);
	WaitForStart_action(N);
END_STEP
TRANSITION FROM WaitForStart TO Seperator := state=2;
END_TRANSITION
STEP Seperator:
END_STEP
TRANSITION FROM Seperator TO Wait_for_Part := Abholpos leer;
END_TRANSITION
TRANSITION FROM Seperator TO SeqEnd := TRUE;
END_TRANSITION
STEP Wait_for_Part:
	Wait_for_Part_entry(P1);
	Wait_for_Part_action(N);
	Wait_for_Part_exit(P0);
END_STEP
TRANSITION FROM Wait_for_Part TO Close_Seperator := Part Ready;
END_TRANSITION
STEP Close_Seperator:
	Close_Seperator_action(N);
END_STEP
TRANSITION FROM Close_Seperator TO Open_Stopper := StateOk;
END_TRANSITION
STEP Open_Stopper: (* min time t#500ms; t#500ms *)
	Open_Stopper_action(N);
END_STEP
TRANSITION FROM Open_Stopper TO Wait_for_Part_ := State Ok;
END_TRANSITION
STEP Wait_for_Part_:
	Wait_for_Part__entry(P1);
	Wait_for_Part__action(N);
	Wait_for_Part__exit(P0);
END_STEP
TRANSITION FROM Wait_for_Part_ TO Close_Stopper := Part Ready;
END_TRANSITION
STEP Close_Stopper: (* min time t#500ms; t#500ms *)
	Close_Stopper_action(N);
END_STEP
TRANSITION FROM Close_Stopper TO Open_Seperator := State Ok;
END_TRANSITION
STEP Open_Seperator:
	Open_Seperator_action(N);
END_STEP
TRANSITION FROM Open_Seperator TO SeqEnd := StateOk;
END_TRANSITION
STEP SeqEnd: (* -> WAIT *)
	SeqEnd_action(N);
END_STEP
TRANSITION FROM SeqEnd TO WaitForStart := TRUE;
END_TRANSITION

ACTION Init_action:
Start:=FALSE;
State:=STATE_WAIT;
MsgOK:=FALSE;
MsgCancel:=FALSE;
SFCRun:=FALSE;
Result:=RESULT_NON;
END_ACTION

ACTION WaitForStart_entry:
State:=STATE_OK;
END_ACTION

ACTION WaitForStart_action:
IF 	Start   THEN
	State:=STATE_RUN;
	Result:=RESULT_NON;
	SFCTimeStart:=TIME();
	Start:=FALSE;
ELSE
	State:=STATE_WAIT;
	MsgOK:=FALSE;
	MsgCancel:=FALSE;
	SFCRun:=FALSE;
END_IF
END_ACTION

ACTION Wait_for_Part_entry:
ProcessMessage01:='';
Delay.IN:=FALSE;
Delay();
END_ACTION

